LIN {X 0,Y 315.723,Z 316.79,A -85,B 0,C 180,E1 -15907.418,E2 -15907.418} C_VEL
LIN {X 0,Y 314.175,Z 327.926,A -85,B 0,C 180,E1 -15908.339,E2 -15908.339} C_VEL
LIN {X 0,Y 312.459,Z 339.529,A -85,B 0,C 180,E1 -15909.595,E2 -15909.595} C_VEL
LIN {X 0,Y 310.609,Z 350.036,A -85,B 0,C 180,E1 -15911.018,E2 -15911.018} C_VEL
LIN {X 0,Y 309.084,Z 358.664,A -85,B 0,C 180,E1 -15912.465,E2 -15912.465} C_VEL
LIN {X 0,Y 307.686,Z 366.655,A -85,B 0,C 180,E1 -15914.091,E2 -15914.091} C_VEL
LIN {X 0,Y 306.274,Z 374.524,A -85,B 0,C 180,E1 -15916.057,E2 -15916.057} C_VEL
LIN {X 0,Y 305.07,Z 380.86,A -85,B 0,C 180,E1 -15918.033,E2 -15918.033} C_VEL
LIN {X 0,Y 304.358,Z 385.924,A -85,B 0,C 180,E1 -15920.026,E2 -15920.026} C_VEL
LIN {X 0,Y 303.916,Z 389.858,A -85,B 0,C 180,E1 -15922.024,E2 -15922.024} C_VEL
LIN {X 0,Y 303.628,Z 393.261,A -85,B 0,C 180,E1 -15924.455,E2 -15924.455} C_VEL
LIN {X 0,Y 303.639,Z 394.706,A -85,B 0,C 180,E1 -15926.018,E2 -15926.018} C_VEL
LIN {X 0,Y 303.654,Z 395.466,A -85,B 0,C 180,E1 -15927.346,E2 -15927.346} C_VEL
LIN {X 0,Y 303.685,Z 395.832,A -85,B 0,C 180,E1 -15928.673,E2 -15928.673} C_VEL
LIN {X 0,Y 303.763,Z 395.804,A -85,B 0,C 180,E1 -15929.999,E2 -15929.999} C_VEL
LIN {X 0,Y 303.694,Z 395.325,A -85,B 0,C 180,E1 -15931.325,E2 -15931.325} C_VEL
LIN {X 0,Y 303.671,Z 394.427,A -85,B 0,C 180,E1 -15932.652,E2 -15932.652} C_VEL
LIN {X 0,Y 303.684,Z 393.121,A -85,B 0,C 180,E1 -15933.98,E2 -15933.98} C_VEL
LIN {X 0,Y 303.668,Z 390.884,A -85,B 0,C 180,E1 -15935.623,E2 -15935.623} C_VEL
LIN {X 0,Y 303.914,Z 386.438,A -85,B 0,C 180,E1 -15937.975,E2 -15937.975} C_VEL
LIN {X 0,Y 304.3,Z 381.396,A -85,B 0,C 180,E1 -15939.974,E2 -15939.974} C_VEL
LIN {X 0,Y 304.898,Z 375.03,A -85,B 0,C 180,E1 -15941.972,E2 -15941.972} C_VEL
LIN {X 0,Y 305.955,Z 367.045,A -85,B 0,C 180,E1 -15943.956,E2 -15943.956} C_VEL
LIN {X 0,Y 306.977,Z 358.879,A -85,B 0,C 180,E1 -15945.604,E2 -15945.604} C_VEL
LIN {X 0,Y 308.137,Z 348.901,A -85,B 0,C 180,E1 -15947.247,E2 -15947.247} C_VEL
LIN {X 0,Y 309.56,Z 337.739,A -85,B 0,C 180,E1 -15948.703,E2 -15948.703} C_VEL
LIN {X 0,Y 310.984,Z 325.048,A -85,B 0,C 180,E1 -15949.987,E2 -15949.987} C_VEL
LIN {X 0,Y 312.215,Z 312.461,A -85,B 0,C 180,E1 -15950.937,E2 -15950.937} C_VEL
LIN {X 0,Y 313.215,Z 299.169,A -85,B 0,C 180,E1 -15951.643,E2 -15951.643} C_VEL
LIN {X 0,Y 313.823,Z 286.404,A -85,B 0,C 180,E1 -15952.074,E2 -15952.074} C_VEL
LIN {X 0,Y 315.222,Z 226.259,A -85,B 0,C 180,E1 -15953.544,E2 -15953.544} C_VEL
LIN {X 0,Y 309.309,Z 183.433,A -85,B 0,C 180,E1 -15955.1,E2 -15955.1} C_VEL
LIN {X 0,Y 309.937,Z 177.619,A -85,B 0,C 180,E1 -15956.605,E2 -15956.605} C_VEL
LIN {X 0,Y 308.248,Z 168.036,A -85,B 0,C 180,E1 -15959.303,E2 -15959.303} C_VEL
LIN {X 0,Y 305.482,Z 155.435,A -85,B 0,C 180,E1 -15963.07,E2 -15963.07} C_VEL
LIN {X 0,Y 305.481,Z 155.431,A -85,B 0,C 180,E1 -15966.738,E2 -15966.738} C_VEL
LIN {X 0,Y 305.455,Z 155.435,A -85,B 0,C 180,E1 -15970.599,E2 -15970.599} C_VEL
LIN {X 0,Y 305.425,Z 155.442,A -85,B 0,C 180,E1 -15973.654,E2 -15973.654} C_VEL
LIN {X 0,Y 305.455,Z 155.436,A -85,B 0,C 180,E1 -15977.413,E2 -15977.413} C_VEL
LIN {X 0,Y 305.475,Z 155.436,A -85,B 0,C 180,E1 -15981.597,E2 -15981.597} C_VEL
LIN {X 0,Y 305.461,Z 155.433,A -85,B 0,C 180,E1 -15984.886,E2 -15984.886} C_VEL
LIN {X 0,Y 305.451,Z 155.434,A -85,B 0,C 180,E1 -15988.354,E2 -15988.354} C_VEL
LIN {X 0,Y 305.52,Z 155.427,A -85,B 0,C 180,E1 -15991.113,E2 -15991.113} C_VEL
LIN {X 0,Y 305.571,Z 155.419,A -85,B 0,C 180,E1 -15994.087,E2 -15994.087} C_VEL
LIN {X 0,Y 305.493,Z 155.429,A -85,B 0,C 180,E1 -15998.402,E2 -15998.402} C_VEL
LIN {X 0,Y 305.541,Z 155.428,A -85,B 0,C 180,E1 -16001.214,E2 -16001.214} C_VEL
LIN {X 0,Y 305.624,Z 155.416,A -85,B 0,C 180,E1 -16005.347,E2 -16005.347} C_VEL
LIN {X 0,Y 305.636,Z 155.412,A -85,B 0,C 180,E1 -16009.399,E2 -16009.399} C_VEL
LIN {X 0,Y 305.806,Z 155.387,A -85,B 0,C 180,E1 -16012.073,E2 -16012.073} C_VEL
LIN {X 0,Y 305.685,Z 155.407,A -85,B 0,C 180,E1 -16014.723,E2 -16014.723} C_VEL
LIN {X 0,Y 305.955,Z 155.375,A -85,B 0,C 180,E1 -16018.683,E2 -16018.683} C_VEL
LIN {X 0,Y 305.955,Z 155.37,A -85,B 0,C 180,E1 -16021.316,E2 -16021.316} C_VEL
LIN {X 0,Y 305.843,Z 155.389,A -85,B 0,C 180,E1 -16026.597,E2 -16026.597} C_VEL
LIN {X 0,Y 305.732,Z 155.399,A -85,B 0,C 180,E1 -16029.259,E2 -16029.259} C_VEL
LIN {X 0,Y 305.585,Z 155.414,A -85,B 0,C 180,E1 -16033.295,E2 -16033.295} C_VEL
LIN {X 0,Y 305.59,Z 155.416,A -85,B 0,C 180,E1 -16036.019,E2 -16036.019} C_VEL
LIN {X 0,Y 305.574,Z 155.418,A -85,B 0,C 180,E1 -16039.445,E2 -16039.445} C_VEL
LIN {X 0,Y 305.487,Z 155.428,A -85,B 0,C 180,E1 -16043.041,E2 -16043.041} C_VEL
LIN {X 0,Y 305.543,Z 155.423,A -85,B 0,C 180,E1 -16046.227,E2 -16046.227} C_VEL
LIN {X 0,Y 305.491,Z 155.428,A -85,B 0,C 180,E1 -16049.049,E2 -16049.049} C_VEL
LIN {X 0,Y 305.44,Z 155.438,A -85,B 0,C 180,E1 -16051.952,E2 -16051.952} C_VEL
LIN {X 0,Y 305.458,Z 155.43,A -85,B 0,C 180,E1 -16055.113,E2 -16055.113} C_VEL
LIN {X 0,Y 305.489,Z 155.429,A -85,B 0,C 180,E1 -16058.539,E2 -16058.539} C_VEL
LIN {X 0,Y 305.517,Z 155.425,A -85,B 0,C 180,E1 -16062.599,E2 -16062.599} C_VEL
LIN {X 0,Y 305.529,Z 155.424,A -85,B 0,C 180,E1 -16066.364,E2 -16066.364} C_VEL
LIN {X 0,Y 305.495,Z 155.433,A -85,B 0,C 180,E1 -16069.899,E2 -16069.899} C_VEL
LIN {X 0,Y 305.497,Z 155.432,A -85,B 0,C 180,E1 -16073.626,E2 -16073.626} C_VEL
LIN {X 0,Y 305.46,Z 155.433,A -85,B 0,C 180,E1 -16076.483,E2 -16076.483} C_VEL
LIN {X 0,Y 305.459,Z 155.438,A -85,B 0,C 180,E1 -16079.591,E2 -16079.591} C_VEL
LIN {X 0,Y 305.516,Z 155.426,A -85,B 0,C 180,E1 -16082.609,E2 -16082.609} C_VEL
LIN {X 0,Y 305.503,Z 155.432,A -85,B 0,C 180,E1 -16085.539,E2 -16085.539} C_VEL
LIN {X 0,Y 305.515,Z 155.428,A -85,B 0,C 180,E1 -16089.816,E2 -16089.816} C_VEL
LIN {X 0,Y 305.57,Z 155.42,A -85,B 0,C 180,E1 -16092.603,E2 -16092.603} C_VEL
LIN {X 0,Y 305.645,Z 155.415,A -85,B 0,C 180,E1 -16095.35,E2 -16095.35} C_VEL
LIN {X 0,Y 305.635,Z 155.415,A -85,B 0,C 180,E1 -16099.4,E2 -16099.4} C_VEL
LIN {X 0,Y 305.809,Z 155.39,A -85,B 0,C 180,E1 -16102.075,E2 -16102.075} C_VEL
LIN {X 0,Y 305.687,Z 155.407,A -85,B 0,C 180,E1 -16104.724,E2 -16104.724} C_VEL
LIN {X 0,Y 305.954,Z 155.374,A -85,B 0,C 180,E1 -16108.685,E2 -16108.685} C_VEL
LIN {X 0,Y 305.954,Z 155.374,A -85,B 0,C 180,E1 -16111.317,E2 -16111.317} C_VEL
LIN {X 0,Y 305.85,Z 155.388,A -85,B 0,C 180,E1 -16116.598,E2 -16116.598} C_VEL
LIN {X 0,Y 305.733,Z 155.401,A -85,B 0,C 180,E1 -16119.261,E2 -16119.261} C_VEL
LIN {X 0,Y 305.646,Z 155.427,A -85,B 0,C 180,E1 -16122.197,E2 -16122.197} C_VEL
LIN {X 0,Y 306.011,Z 157.364,A -85,B 0,C 180,E1 -16122.772,E2 -16122.772} C_VEL
LIN {X 0,Y 314.604,Z 181.076,A -85,B 0,C 180,E1 -16124.022,E2 -16124.022} C_VEL
LIN {X 0,Y 316.001,Z 185.936,A -85,B 0,C 180,E1 -16124.243,E2 -16124.243} C_VEL
LIN {X 0,Y 313.909,Z 265.333,A -85,B 0,C 180,E1 -16126.208,E2 -16126.208} C_VEL
LIN {X 0,Y 313.17,Z 279.059,A -85,B 0,C 180,E1 -16126.82,E2 -16126.82} C_VEL
LIN {X 0,Y 312.365,Z 291.964,A -85,B 0,C 180,E1 -16127.683,E2 -16127.683} C_VEL
LIN {X 0,Y 311.294,Z 304.537,A -85,B 0,C 180,E1 -16128.822,E2 -16128.822} C_VEL
LIN {X 0,Y 310.107,Z 315.16,A -85,B 0,C 180,E1 -16130.047,E2 -16130.047} C_VEL
LIN {X 0,Y 308.85,Z 325.402,A -85,B 0,C 180,E1 -16131.527,E2 -16131.527} C_VEL
LIN {X 0,Y 307.7,Z 334.503,A -85,B 0,C 180,E1 -16133.154,E2 -16133.154} C_VEL
LIN {X 0,Y 306.538,Z 343.308,A -85,B 0,C 180,E1 -16135.098,E2 -16135.098} C_VEL
LIN {X 0,Y 305.712,Z 349.648,A -85,B 0,C 180,E1 -16136.832,E2 -16136.832} C_VEL
LIN {X 0,Y 304.919,Z 355.858,A -85,B 0,C 180,E1 -16138.949,E2 -16138.949} C_VEL
LIN {X 0,Y 304.31,Z 361.08,A -85,B 0,C 180,E1 -16141.296,E2 -16141.296} C_VEL
LIN {X 0,Y 303.83,Z 364.938,A -85,B 0,C 180,E1 -16143.722,E2 -16143.722} C_VEL
LIN {X 0,Y 303.556,Z 367.113,A -85,B 0,C 180,E1 -16145.873,E2 -16145.873} C_VEL
LIN {X 0,Y 303.487,Z 368.209,A -85,B 0,C 180,E1 -16148.062,E2 -16148.062} C_VEL
LIN {X 0,Y 303.613,Z 368.161,A -85,B 0,C 180,E1 -16150.403,E2 -16150.403} C_VEL
LIN {X 0,Y 303.887,Z 367.26,A -85,B 0,C 180,E1 -16152.264,E2 -16152.264} C_VEL
LIN {X 0,Y 304.351,Z 365.346,A -85,B 0,C 180,E1 -16154.289,E2 -16154.289} C_VEL
LIN {X 0,Y 305.116,Z 361.546,A -85,B 0,C 180,E1 -16156.803,E2 -16156.803} C_VEL
LIN {X 0,Y 306.252,Z 356.287,A -85,B 0,C 180,E1 -16159.228,E2 -16159.228} C_VEL
LIN {X 0,Y 307.557,Z 349.621,A -85,B 0,C 180,E1 -16161.505,E2 -16161.505} C_VEL
LIN {X 0,Y 308.904,Z 342.905,A -85,B 0,C 180,E1 -16163.32,E2 -16163.32} C_VEL
LIN {X 0,Y 310.53,Z 334.566,A -85,B 0,C 180,E1 -16165.141,E2 -16165.141} C_VEL
LIN {X 0,Y 312.217,Z 325.27,A -85,B 0,C 180,E1 -16166.776,E2 -16166.776} C_VEL
LIN {X 0,Y 313.93,Z 314.467,A -85,B 0,C 180,E1 -16168.291,E2 -16168.291} C_VEL
LIN {X 0,Y 315.533,Z 303.485,A -85,B 0,C 180,E1 -16169.507,E2 -16169.507} C_VEL
LIN {X 0,Y 315.612,Z 298.386,A -85,B 0,C 180,E1 -16170.05,E2 -16170.05} C_VEL
LIN {X 0,Y 314.022,Z 290.018,A -85,B 0,C 180,E1 -16170.973,E2 -16170.973} C_VEL
LIN {X 0,Y 312.204,Z 281.348,A -85,B 0,C 180,E1 -16171.781,E2 -16171.781} C_VEL
LIN {X 0,Y 311.905,Z 275.779,A -85,B 0,C 180,E1 -16172.133,E2 -16172.133} C_VEL
LIN {X 0,Y 312.55,Z 264.777,A -85,B 0,C 180,E1 -16172.574,E2 -16172.574} C_VEL
LIN {X 0,Y 315.135,Z 192.637,A -85,B 0,C 180,E1 -16174.416,E2 -16174.416} C_VEL
LIN {X 0,Y 308.893,Z 177.993,A -85,B 0,C 180,E1 -16175.583,E2 -16175.583} C_VEL
LIN {X 0,Y 302.671,Z 165.931,A -85,B 0,C 180,E1 -16176.751,E2 -16176.751} C_VEL
LIN {X 0,Y 299.317,Z 159.58,A -85,B 0,C 180,E1 -16177.435,E2 -16177.435} C_VEL
LIN {X 0,Y 298.422,Z 156.314,A -85,B 0,C 180,E1 -16178.772,E2 -16178.772} C_VEL
LIN {X 0,Y 298.507,Z 156.301,A -85,B 0,C 180,E1 -16182.178,E2 -16182.178} C_VEL
LIN {X 0,Y 298.589,Z 156.293,A -85,B 0,C 180,E1 -16184.995,E2 -16184.995} C_VEL
LIN {X 0,Y 298.587,Z 156.292,A -85,B 0,C 180,E1 -16189.147,E2 -16189.147} C_VEL
LIN {X 0,Y 298.702,Z 156.279,A -85,B 0,C 180,E1 -16191.885,E2 -16191.885} C_VEL
LIN {X 0,Y 298.633,Z 156.287,A -85,B 0,C 180,E1 -16194.599,E2 -16194.599} C_VEL
LIN {X 0,Y 298.908,Z 156.245,A -85,B 0,C 180,E1 -16198.653,E2 -16198.653} C_VEL
LIN {X 0,Y 298.907,Z 156.252,A -85,B 0,C 180,E1 -16201.348,E2 -16201.348} C_VEL
LIN {X 0,Y 298.74,Z 156.26,A -85,B 0,C 180,E1 -16206.756,E2 -16206.756} C_VEL
LIN {X 0,Y 298.629,Z 156.286,A -85,B 0,C 180,E1 -16209.483,E2 -16209.483} C_VEL
LIN {X 0,Y 298.513,Z 156.299,A -85,B 0,C 180,E1 -16213.618,E2 -16213.618} C_VEL
LIN {X 0,Y 298.438,Z 156.306,A -85,B 0,C 180,E1 -16216.416,E2 -16216.416} C_VEL
LIN {X 0,Y 298.426,Z 156.301,A -85,B 0,C 180,E1 -16219.606,E2 -16219.606} C_VEL
LIN {X 0,Y 298.384,Z 156.307,A -85,B 0,C 180,E1 -16223.605,E2 -16223.605} C_VEL
LIN {X 0,Y 298.406,Z 156.312,A -85,B 0,C 180,E1 -16226.583,E2 -16226.583} C_VEL
LIN {X 0,Y 298.362,Z 156.32,A -85,B 0,C 180,E1 -16229.648,E2 -16229.648} C_VEL
LIN {X 0,Y 298.398,Z 156.313,A -85,B 0,C 180,E1 -16232.801,E2 -16232.801} C_VEL
LIN {X 0,Y 298.446,Z 156.311,A -85,B 0,C 180,E1 -16236.806,E2 -16236.806} C_VEL
LIN {X 0,Y 298.353,Z 156.317,A -85,B 0,C 180,E1 -16241.079,E2 -16241.079} C_VEL
LIN {X 0,Y 298.36,Z 156.325,A -85,B 0,C 180,E1 -16245.035,E2 -16245.035} C_VEL
LIN {X 0,Y 298.353,Z 156.322,A -85,B 0,C 180,E1 -16248.921,E2 -16248.921} C_VEL
LIN {X 0,Y 298.443,Z 156.429,A -85,B 0,C 180,E1 -16252.981,E2 -16252.981} C_VEL
LIN {X 0,Y 300.851,Z 165.427,A -85,B 0,C 180,E1 -16256.251,E2 -16256.251} C_VEL
LIN {X 0,Y 303.031,Z 174.547,A -85,B 0,C 180,E1 -16259.32,E2 -16259.32} C_VEL
LIN {X 0,Y 304.282,Z 180.764,A -85,B 0,C 180,E1 -16261.284,E2 -16261.284} C_VEL
LIN {X 0,Y 307.064,Z 187.661,A -85,B 0,C 180,E1 -16261.845,E2 -16261.845} C_VEL
LIN {X 0,Y 310.502,Z 204.648,A -85,B 0,C 180,E1 -16262.771,E2 -16262.771} C_VEL
LIN {X 0,Y 313.101,Z 221.424,A -85,B 0,C 180,E1 -16263.561,E2 -16263.561} C_VEL
LIN {X 0,Y 313.982,Z 230.204,A -85,B 0,C 180,E1 -16263.914,E2 -16263.914} C_VEL
LIN {X 0,Y 311.806,Z 291.118,A -85,B 0,C 180,E1 -16265.488,E2 -16265.488} C_VEL
LIN {X 0,Y 310.703,Z 305.109,A -85,B 0,C 180,E1 -16266.106,E2 -16266.106} C_VEL
LIN {X 0,Y 309.231,Z 317.646,A -85,B 0,C 180,E1 -16266.917,E2 -16266.917} C_VEL
LIN {X 0,Y 307.45,Z 330.063,A -85,B 0,C 180,E1 -16268.017,E2 -16268.017} C_VEL
LIN {X 0,Y 305.641,Z 341.228,A -85,B 0,C 180,E1 -16269.295,E2 -16269.295} C_VEL
LIN {X 0,Y 303.751,Z 351.344,A -85,B 0,C 180,E1 -16270.748,E2 -16270.748} C_VEL
LIN {X 0,Y 302.012,Z 360.519,A -85,B 0,C 180,E1 -16272.39,E2 -16272.39} C_VEL
LIN {X 0,Y 300.33,Z 369.507,A -85,B 0,C 180,E1 -16274.388,E2 -16274.388} C_VEL
LIN {X 0,Y 298.93,Z 376.767,A -85,B 0,C 180,E1 -16276.401,E2 -16276.401} C_VEL
LIN {X 0,Y 297.828,Z 382.586,A -85,B 0,C 180,E1 -16278.428,E2 -16278.428} C_VEL
LIN {X 0,Y 297.139,Z 387.208,A -85,B 0,C 180,E1 -16280.469,E2 -16280.469} C_VEL
LIN {X 0,Y 296.713,Z 390.748,A -85,B 0,C 180,E1 -16282.514,E2 -16282.514} C_VEL
LIN {X 0,Y 296.535,Z 393.286,A -85,B 0,C 180,E1 -16284.559,E2 -16284.559} C_VEL
LIN {X 0,Y 296.535,Z 394.428,A -85,B 0,C 180,E1 -16285.922,E2 -16285.922} C_VEL
LIN {X 0,Y 296.577,Z 395.17,A -85,B 0,C 180,E1 -16287.283,E2 -16287.283} C_VEL
LIN {X 0,Y 296.598,Z 395.515,A -85,B 0,C 180,E1 -16288.641,E2 -16288.641} C_VEL
LIN {X 0,Y 296.671,Z 395.458,A -85,B 0,C 180,E1 -16289.999,E2 -16289.999} C_VEL
LIN {X 0,Y 296.606,Z 394.943,A -85,B 0,C 180,E1 -16291.357,E2 -16291.357} C_VEL
LIN {X 0,Y 296.594,Z 394.023,A -85,B 0,C 180,E1 -16292.716,E2 -16292.716} C_VEL
LIN {X 0,Y 296.597,Z 392.694,A -85,B 0,C 180,E1 -16294.076,E2 -16294.076} C_VEL
LIN {X 0,Y 296.616,Z 389.835,A -85,B 0,C 180,E1 -16296.119,E2 -16296.119} C_VEL
LIN {X 0,Y 296.85,Z 385.909,A -85,B 0,C 180,E1 -16298.166,E2 -16298.166} C_VEL
LIN {X 0,Y 297.361,Z 379.828,A -85,B 0,C 180,E1 -16300.554,E2 -16300.554} C_VEL
LIN {X 0,Y 298.121,Z 373.12,A -85,B 0,C 180,E1 -16302.594,E2 -16302.594} C_VEL
LIN {X 0,Y 299.207,Z 364.774,A -85,B 0,C 180,E1 -16304.625,E2 -16304.625} C_VEL
LIN {X 0,Y 300.338,Z 355.816,A -85,B 0,C 180,E1 -16306.378,E2 -16306.378} C_VEL
LIN {X 0,Y 301.696,Z 345.618,A -85,B 0,C 180,E1 -16307.978,E2 -16307.978} C_VEL
LIN {X 0,Y 303.163,Z 333.703,A -85,B 0,C 180,E1 -16309.465,E2 -16309.465} C_VEL
LIN {X 0,Y 304.557,Z 321.737,A -85,B 0,C 180,E1 -16310.603,E2 -16310.603} C_VEL
LIN {X 0,Y 305.703,Z 309.357,A -85,B 0,C 180,E1 -16311.493,E2 -16311.493} C_VEL
LIN {X 0,Y 306.562,Z 296.715,A -85,B 0,C 180,E1 -16312.137,E2 -16312.137} C_VEL
LIN {X 0,Y 307.169,Z 282.226,A -85,B 0,C 180,E1 -16312.578,E2 -16312.578} C_VEL
LIN {X 0,Y 308.452,Z 226.602,A -85,B 0,C 180,E1 -16313.972,E2 -16313.972} C_VEL
LIN {X 0,Y 302.488,Z 183.168,A -85,B 0,C 180,E1 -16315.59,E2 -16315.59} C_VEL
LIN {X 0,Y 302.925,Z 178.248,A -85,B 0,C 180,E1 -16316.897,E2 -16316.897} C_VEL
LIN {X 0,Y 300.938,Z 167.767,A -85,B 0,C 180,E1 -16319.946,E2 -16319.946} C_VEL
LIN {X 0,Y 298.431,Z 156.313,A -85,B 0,C 180,E1 -16323.449,E2 -16323.449} C_VEL
LIN {X 0,Y 298.451,Z 156.307,A -85,B 0,C 180,E1 -16326.808,E2 -16326.808} C_VEL
LIN {X 0,Y 298.409,Z 156.314,A -85,B 0,C 180,E1 -16329.485,E2 -16329.485} C_VEL
LIN {X 0,Y 298.399,Z 156.314,A -85,B 0,C 180,E1 -16333.102,E2 -16333.102} C_VEL
LIN {X 0,Y 298.403,Z 156.312,A -85,B 0,C 180,E1 -16336.92,E2 -16336.92} C_VEL
LIN {X 0,Y 298.404,Z 156.313,A -85,B 0,C 180,E1 -16341.005,E2 -16341.005} C_VEL
LIN {X 0,Y 298.418,Z 156.313,A -85,B 0,C 180,E1 -16343.929,E2 -16343.929} C_VEL
LIN {X 0,Y 298.394,Z 156.315,A -85,B 0,C 180,E1 -16347.982,E2 -16347.982} C_VEL
LIN {X 0,Y 298.469,Z 156.305,A -85,B 0,C 180,E1 -16351.904,E2 -16351.904} C_VEL
LIN {X 0,Y 298.485,Z 156.303,A -85,B 0,C 180,E1 -16354.923,E2 -16354.923} C_VEL
LIN {X 0,Y 298.437,Z 156.313,A -85,B 0,C 180,E1 -16359.314,E2 -16359.314} C_VEL
LIN {X 0,Y 298.476,Z 156.302,A -85,B 0,C 180,E1 -16362.175,E2 -16362.175} C_VEL
LIN {X 0,Y 298.584,Z 156.291,A -85,B 0,C 180,E1 -16364.994,E2 -16364.994} C_VEL
LIN {X 0,Y 298.592,Z 156.292,A -85,B 0,C 180,E1 -16369.146,E2 -16369.146} C_VEL
LIN {X 0,Y 298.752,Z 156.265,A -85,B 0,C 180,E1 -16371.885,E2 -16371.885} C_VEL
LIN {X 0,Y 298.656,Z 156.281,A -85,B 0,C 180,E1 -16374.598,E2 -16374.598} C_VEL
LIN {X 0,Y 298.922,Z 156.25,A -85,B 0,C 180,E1 -16378.652,E2 -16378.652} C_VEL
LIN {X 0,Y 298.921,Z 156.245,A -85,B 0,C 180,E1 -16381.346,E2 -16381.346} C_VEL
LIN {X 0,Y 298.789,Z 156.269,A -85,B 0,C 180,E1 -16386.753,E2 -16386.753} C_VEL
LIN {X 0,Y 298.677,Z 156.277,A -85,B 0,C 180,E1 -16389.48,E2 -16389.48} C_VEL
LIN {X 0,Y 298.548,Z 156.289,A -85,B 0,C 180,E1 -16393.615,E2 -16393.615} C_VEL
LIN {X 0,Y 298.545,Z 156.296,A -85,B 0,C 180,E1 -16396.408,E2 -16396.408} C_VEL
LIN {X 0,Y 298.508,Z 156.299,A -85,B 0,C 180,E1 -16399.655,E2 -16399.655} C_VEL
LIN {X 0,Y 298.454,Z 156.304,A -85,B 0,C 180,E1 -16403.597,E2 -16403.597} C_VEL
LIN {X 0,Y 298.485,Z 156.302,A -85,B 0,C 180,E1 -16406.574,E2 -16406.574} C_VEL
LIN {X 0,Y 298.416,Z 156.31,A -85,B 0,C 180,E1 -16409.641,E2 -16409.641} C_VEL
LIN {X 0,Y 298.391,Z 156.312,A -85,B 0,C 180,E1 -16412.8,E2 -16412.8} C_VEL
LIN {X 0,Y 298.465,Z 156.301,A -85,B 0,C 180,E1 -16416.814,E2 -16416.814} C_VEL
LIN {X 0,Y 298.452,Z 156.305,A -85,B 0,C 180,E1 -16421.249,E2 -16421.249} C_VEL
LIN {X 0,Y 298.484,Z 156.299,A -85,B 0,C 180,E1 -16425.061,E2 -16425.061} C_VEL
LIN {X 0,Y 298.451,Z 156.305,A -85,B 0,C 180,E1 -16428.897,E2 -16428.897} C_VEL
LIN {X 0,Y 298.465,Z 156.304,A -85,B 0,C 180,E1 -16433.186,E2 -16433.186} C_VEL
LIN {X 0,Y 298.39,Z 156.314,A -85,B 0,C 180,E1 -16437.2,E2 -16437.2} C_VEL
LIN {X 0,Y 298.427,Z 156.309,A -85,B 0,C 180,E1 -16440.615,E2 -16440.615} C_VEL
LIN {X 0,Y 298.479,Z 156.307,A -85,B 0,C 180,E1 -16443.474,E2 -16443.474} C_VEL
LIN {X 0,Y 298.43,Z 156.309,A -85,B 0,C 180,E1 -16446.698,E2 -16446.698} C_VEL
LIN {X 0,Y 298.535,Z 156.296,A -85,B 0,C 180,E1 -16450.757,E2 -16450.757} C_VEL
LIN {X 0,Y 298.589,Z 156.292,A -85,B 0,C 180,E1 -16454.995,E2 -16454.995} C_VEL
LIN {X 0,Y 298.59,Z 156.294,A -85,B 0,C 180,E1 -16459.147,E2 -16459.147} C_VEL
LIN {X 0,Y 298.754,Z 156.269,A -85,B 0,C 180,E1 -16461.887,E2 -16461.887} C_VEL
LIN {X 0,Y 298.657,Z 156.282,A -85,B 0,C 180,E1 -16464.6,E2 -16464.6} C_VEL
LIN {X 0,Y 298.92,Z 156.25,A -85,B 0,C 180,E1 -16468.654,E2 -16468.654} C_VEL
LIN {X 0,Y 298.921,Z 156.25,A -85,B 0,C 180,E1 -16471.348,E2 -16471.348} C_VEL
LIN {X 0,Y 298.795,Z 156.268,A -85,B 0,C 180,E1 -16476.755,E2 -16476.755} C_VEL
LIN {X 0,Y 298.678,Z 156.28,A -85,B 0,C 180,E1 -16479.481,E2 -16479.481} C_VEL
LIN {X 0,Y 298.604,Z 156.465,A -85,B 0,C 180,E1 -16481.885,E2 -16481.885} C_VEL
LIN {X 0,Y 298.907,Z 157.765,A -85,B 0,C 180,E1 -16482.239,E2 -16482.239} C_VEL
LIN {X 0,Y 307.692,Z 181.814,A -85,B 0,C 180,E1 -16483.559,E2 -16483.559} C_VEL
LIN {X 0,Y 309.444,Z 187.449,A -85,B 0,C 180,E1 -16483.834,E2 -16483.834} C_VEL
LIN {X 0,Y 307.204,Z 264.994,A -85,B 0,C 180,E1 -16485.781,E2 -16485.781} C_VEL
LIN {X 0,Y 306.438,Z 278.893,A -85,B 0,C 180,E1 -16486.403,E2 -16486.403} C_VEL
LIN {X 0,Y 305.639,Z 291.188,A -85,B 0,C 180,E1 -16487.222,E2 -16487.222} C_VEL
LIN {X 0,Y 304.6,Z 303.395,A -85,B 0,C 180,E1 -16488.323,E2 -16488.323} C_VEL
LIN {X 0,Y 303.316,Z 314.744,A -85,B 0,C 180,E1 -16489.633,E2 -16489.633} C_VEL
LIN {X 0,Y 302.094,Z 324.416,A -85,B 0,C 180,E1 -16491.023,E2 -16491.023} C_VEL
LIN {X 0,Y 300.886,Z 333.684,A -85,B 0,C 180,E1 -16492.67,E2 -16492.67} C_VEL
LIN {X 0,Y 299.66,Z 342.905,A -85,B 0,C 180,E1 -16494.712,E2 -16494.712} C_VEL
LIN {X 0,Y 298.721,Z 349.824,A -85,B 0,C 180,E1 -16496.619,E2 -16496.619} C_VEL
LIN {X 0,Y 297.919,Z 355.737,A -85,B 0,C 180,E1 -16498.649,E2 -16498.649} C_VEL
LIN {X 0,Y 297.369,Z 360.088,A -85,B 0,C 180,E1 -16500.54,E2 -16500.54} C_VEL
LIN {X 0,Y 296.875,Z 364.287,A -85,B 0,C 180,E1 -16502.99,E2 -16502.99} C_VEL
LIN {X 0,Y 296.568,Z 366.335,A -85,B 0,C 180,E1 -16504.664,E2 -16504.664} C_VEL
LIN {X 0,Y 296.438,Z 367.717,A -85,B 0,C 180,E1 -16506.35,E2 -16506.35} C_VEL
LIN {X 0,Y 296.418,Z 368.595,A -85,B 0,C 180,E1 -16508.519,E2 -16508.519} C_VEL
LIN {X 0,Y 296.556,Z 368.451,A -85,B 0,C 180,E1 -16510.682,E2 -16510.682} C_VEL
LIN {X 0,Y 297.028,Z 366.898,A -85,B 0,C 180,E1 -16513.329,E2 -16513.329} C_VEL
LIN {X 0,Y 297.792,Z 363.71,A -85,B 0,C 180,E1 -16515.987,E2 -16515.987} C_VEL
LIN {X 0,Y 298.498,Z 360.434,A -85,B 0,C 180,E1 -16517.874,E2 -16517.874} C_VEL
LIN {X 0,Y 299.642,Z 355.066,A -85,B 0,C 180,E1 -16520.188,E2 -16520.188} C_VEL
LIN {X 0,Y 300.861,Z 349.567,A -85,B 0,C 180,E1 -16522.036,E2 -16522.036} C_VEL
LIN {X 0,Y 302.431,Z 342.185,A -85,B 0,C 180,E1 -16524.031,E2 -16524.031} C_VEL
LIN {X 0,Y 304.025,Z 334.282,A -85,B 0,C 180,E1 -16525.754,E2 -16525.754} C_VEL
LIN {X 0,Y 305.882,Z 324.255,A -85,B 0,C 180,E1 -16527.505,E2 -16527.505} C_VEL
LIN {X 0,Y 307.509,Z 314.576,A -85,B 0,C 180,E1 -16528.865,E2 -16528.865} C_VEL
LIN {X 0,Y 309.289,Z 302.642,A -85,B 0,C 180,E1 -16530.195,E2 -16530.195} C_VEL
LIN {X 0,Y 310.73,Z 289.888,A -85,B 0,C 180,E1 -16531.275,E2 -16531.275} C_VEL
LIN {X 0,Y 311.787,Z 277.709,A -85,B 0,C 180,E1 -16532.034,E2 -16532.034} C_VEL
LIN {X 0,Y 311.905,Z 275.779,A -85,B 0,C 180,E1 -16532.133,E2 -16532.133} C_VEL
LIN {X 0,Y 311.619,Z 270.11,A -85,B 0,C 180,E1 -16532.451,E2 -16532.451} C_VEL
LIN {X 0,Y 307.508,Z 252.608,A -85,B 0,C 180,E1 -16533.498,E2 -16533.498} C_VEL
LIN {X 0,Y 307.059,Z 247.821,A -85,B 0,C 180,E1 -16533.684,E2 -16533.684} C_VEL
LIN {X 0,Y 307.104,Z 245.879,A -85,B 0,C 180,E1 -16533.736,E2 -16533.736} C_VEL
LIN {X 0,Y 309.095,Z 194.644,A -85,B 0,C 180,E1 -16535.05,E2 -16535.05} C_VEL
LIN {X 0,Y 302.855,Z 180.204,A -85,B 0,C 180,E1 -16536.272,E2 -16536.272} C_VEL
LIN {X 0,Y 297.115,Z 169.053,A -85,B 0,C 180,E1 -16537.402,E2 -16537.402} C_VEL
LIN {X 0,Y 292.177,Z 160.065,A -85,B 0,C 180,E1 -16538.435,E2 -16538.435} C_VEL
LIN {X 0,Y 291.398,Z 157.19,A -85,B 0,C 180,E1 -16539.633,E2 -16539.633} C_VEL
LIN {X 0,Y 291.444,Z 157.183,A -85,B 0,C 180,E1 -16543.18,E2 -16543.18} C_VEL
LIN {X 0,Y 291.519,Z 157.177,A -85,B 0,C 180,E1 -16546.05,E2 -16546.05} C_VEL
LIN {X 0,Y 291.572,Z 157.167,A -85,B 0,C 180,E1 -16550.287,E2 -16550.287} C_VEL
LIN {X 0,Y 291.691,Z 157.151,A -85,B 0,C 180,E1 -16553.082,E2 -16553.082} C_VEL
LIN {X 0,Y 291.875,Z 157.121,A -85,B 0,C 180,E1 -16558.621,E2 -16558.621} C_VEL
LIN {X 0,Y 291.874,Z 157.128,A -85,B 0,C 180,E1 -16561.381,E2 -16561.381} C_VEL
LIN {X 0,Y 291.692,Z 157.138,A -85,B 0,C 180,E1 -16566.92,E2 -16566.92} C_VEL
LIN {X 0,Y 291.572,Z 157.161,A -85,B 0,C 180,E1 -16569.715,E2 -16569.715} C_VEL
LIN {X 0,Y 291.476,Z 157.172,A -85,B 0,C 180,E1 -16573.953,E2 -16573.953} C_VEL
LIN {X 0,Y 291.392,Z 157.185,A -85,B 0,C 180,E1 -16576.824,E2 -16576.824} C_VEL
LIN {X 0,Y 291.368,Z 157.181,A -85,B 0,C 180,E1 -16579.827,E2 -16579.827} C_VEL
LIN {X 0,Y 291.328,Z 157.187,A -85,B 0,C 180,E1 -16584.212,E2 -16584.212} C_VEL
LIN {X 0,Y 291.333,Z 157.187,A -85,B 0,C 180,E1 -16587.281,E2 -16587.281} C_VEL
LIN {X 0,Y 291.307,Z 157.197,A -85,B 0,C 180,E1 -16590.441,E2 -16590.441} C_VEL
LIN {X 0,Y 291.349,Z 157.193,A -85,B 0,C 180,E1 -16593.699,E2 -16593.699} C_VEL
LIN {X 0,Y 291.372,Z 157.189,A -85,B 0,C 180,E1 -16597.251,E2 -16597.251} C_VEL
LIN {X 0,Y 291.304,Z 157.197,A -85,B 0,C 180,E1 -16600.648,E2 -16600.648} C_VEL
LIN {X 0,Y 291.286,Z 157.201,A -85,B 0,C 180,E1 -16604.404,E2 -16604.404} C_VEL
LIN {X 0,Y 291.3,Z 157.202,A -85,B 0,C 180,E1 -16608.411,E2 -16608.411} C_VEL
LIN {X 0,Y 291.358,Z 157.293,A -85,B 0,C 180,E1 -16612.071,E2 -16612.071} C_VEL
LIN {X 0,Y 293.771,Z 165.928,A -85,B 0,C 180,E1 -16615.376,E2 -16615.376} C_VEL
LIN {X 0,Y 296.255,Z 176.398,A -85,B 0,C 180,E1 -16619.035,E2 -16619.035} C_VEL
LIN {X 0,Y 297.101,Z 180.321,A -85,B 0,C 180,E1 -16620.32,E2 -16620.32} C_VEL
LIN {X 0,Y 301.44,Z 190.585,A -85,B 0,C 180,E1 -16621.231,E2 -16621.231} C_VEL
LIN {X 0,Y 304.613,Z 206.594,A -85,B 0,C 180,E1 -16622.134,E2 -16622.134} C_VEL
LIN {X 0,Y 307.117,Z 223.332,A -85,B 0,C 180,E1 -16622.942,E2 -16622.942} C_VEL
LIN {X 0,Y 307.888,Z 231.171,A -85,B 0,C 180,E1 -16623.265,E2 -16623.265} C_VEL
LIN {X 0,Y 305.646,Z 290.506,A -85,B 0,C 180,E1 -16624.824,E2 -16624.824} C_VEL
LIN {X 0,Y 304.485,Z 304.521,A -85,B 0,C 180,E1 -16625.45,E2 -16625.45} C_VEL
LIN {X 0,Y 303.029,Z 316.591,A -85,B 0,C 180,E1 -16626.235,E2 -16626.235} C_VEL
LIN {X 0,Y 301.1,Z 329.132,A -85,B 0,C 180,E1 -16627.347,E2 -16627.347} C_VEL
LIN {X 0,Y 299.229,Z 340.365,A -85,B 0,C 180,E1 -16628.65,E2 -16628.65} C_VEL
LIN {X 0,Y 297.226,Z 350.59,A -85,B 0,C 180,E1 -16630.128,E2 -16630.128} C_VEL
LIN {X 0,Y 295.239,Z 360.661,A -85,B 0,C 180,E1 -16631.973,E2 -16631.973} C_VEL
LIN {X 0,Y 293.458,Z 369.574,A -85,B 0,C 180,E1 -16634.013,E2 -16634.013} C_VEL
LIN {X 0,Y 292.006,Z 376.739,A -85,B 0,C 180,E1 -16636.072,E2 -16636.072} C_VEL
LIN {X 0,Y 290.843,Z 382.495,A -85,B 0,C 180,E1 -16638.146,E2 -16638.146} C_VEL
LIN {X 0,Y 290.108,Z 387.056,A -85,B 0,C 180,E1 -16640.236,E2 -16640.236} C_VEL
LIN {X 0,Y 289.817,Z 389.483,A -85,B 0,C 180,E1 -16641.633,E2 -16641.633} C_VEL
LIN {X 0,Y 289.57,Z 391.478,A -85,B 0,C 180,E1 -16643.029,E2 -16643.029} C_VEL
LIN {X 0,Y 289.441,Z 393.176,A -85,B 0,C 180,E1 -16644.588,E2 -16644.588} C_VEL
LIN {X 0,Y 289.499,Z 394.874,A -85,B 0,C 180,E1 -16647.216,E2 -16647.216} C_VEL
LIN {X 0,Y 289.513,Z 395.199,A -85,B 0,C 180,E1 -16648.608,E2 -16648.608} C_VEL
LIN {X 0,Y 289.581,Z 395.103,A -85,B 0,C 180,E1 -16649.999,E2 -16649.999} C_VEL
LIN {X 0,Y 289.521,Z 394.562,A -85,B 0,C 180,E1 -16651.39,E2 -16651.39} C_VEL
LIN {X 0,Y 289.519,Z 393.62,A -85,B 0,C 180,E1 -16652.782,E2 -16652.782} C_VEL
LIN {X 0,Y 289.512,Z 392.266,A -85,B 0,C 180,E1 -16654.176,E2 -16654.176} C_VEL
LIN {X 0,Y 289.555,Z 389.359,A -85,B 0,C 180,E1 -16656.27,E2 -16656.27} C_VEL
LIN {X 0,Y 289.781,Z 385.379,A -85,B 0,C 180,E1 -16658.366,E2 -16658.366} C_VEL
LIN {X 0,Y 290.332,Z 379.211,A -85,B 0,C 180,E1 -16660.812,E2 -16660.812} C_VEL
LIN {X 0,Y 291.173,Z 372.439,A -85,B 0,C 180,E1 -16662.9,E2 -16662.9} C_VEL
LIN {X 0,Y 292.317,Z 364.015,A -85,B 0,C 180,E1 -16664.978,E2 -16664.978} C_VEL
LIN {X 0,Y 293.426,Z 355.317,A -85,B 0,C 180,E1 -16666.703,E2 -16666.703} C_VEL
LIN {X 0,Y 294.842,Z 344.593,A -85,B 0,C 180,E1 -16668.41,E2 -16668.41} C_VEL
LIN {X 0,Y 296.237,Z 333.98,A -85,B 0,C 180,E1 -16669.759,E2 -16669.759} C_VEL
LIN {X 0,Y 297.677,Z 322.234,A -85,B 0,C 180,E1 -16670.921,E2 -16670.921} C_VEL
LIN {X 0,Y 298.844,Z 310.095,A -85,B 0,C 180,E1 -16671.83,E2 -16671.83} C_VEL
LIN {X 0,Y 299.773,Z 297.017,A -85,B 0,C 180,E1 -16672.529,E2 -16672.529} C_VEL
LIN {X 0,Y 300.419,Z 283.01,A -85,B 0,C 180,E1 -16672.978,E2 -16672.978} C_VEL
LIN {X 0,Y 301.746,Z 227.294,A -85,B 0,C 180,E1 -16674.409,E2 -16674.409} C_VEL
LIN {X 0,Y 295.685,Z 182.895,A -85,B 0,C 180,E1 -16676.1,E2 -16676.1} C_VEL
LIN {X 0,Y 295.987,Z 180.255,A -85,B 0,C 180,E1 -16676.816,E2 -16676.816} C_VEL
LIN {X 0,Y 294.589,Z 171.875,A -85,B 0,C 180,E1 -16679.278,E2 -16679.278} C_VEL
LIN {X 0,Y 291.962,Z 159.672,A -85,B 0,C 180,E1 -16683.047,E2 -16683.047} C_VEL
LIN {X 0,Y 291.382,Z 157.19,A -85,B 0,C 180,E1 -16683.894,E2 -16683.894} C_VEL
LIN {X 0,Y 291.385,Z 157.188,A -85,B 0,C 180,E1 -16687.255,E2 -16687.255} C_VEL
LIN {X 0,Y 291.334,Z 157.195,A -85,B 0,C 180,E1 -16690.641,E2 -16690.641} C_VEL
LIN {X 0,Y 291.29,Z 157.2,A -85,B 0,C 180,E1 -16694.401,E2 -16694.401} C_VEL
LIN {X 0,Y 291.326,Z 157.194,A -85,B 0,C 180,E1 -16698.403,E2 -16698.403} C_VEL
LIN {X 0,Y 291.353,Z 157.192,A -85,B 0,C 180,E1 -16701.157,E2 -16701.157} C_VEL
LIN {X 0,Y 291.36,Z 157.19,A -85,B 0,C 180,E1 -16704.625,E2 -16704.625} C_VEL
LIN {X 0,Y 291.371,Z 157.19,A -85,B 0,C 180,E1 -16707.95,E2 -16707.95} C_VEL
LIN {X 0,Y 291.384,Z 157.187,A -85,B 0,C 180,E1 -16711.158,E2 -16711.158} C_VEL
LIN {X 0,Y 291.419,Z 157.182,A -85,B 0,C 180,E1 -16714.271,E2 -16714.271} C_VEL
LIN {X 0,Y 291.378,Z 157.19,A -85,B 0,C 180,E1 -16717.299,E2 -16717.299} C_VEL
LIN {X 0,Y 291.456,Z 157.177,A -85,B 0,C 180,E1 -16720.269,E2 -16720.269} C_VEL
LIN {X 0,Y 291.495,Z 157.171,A -85,B 0,C 180,E1 -16724.664,E2 -16724.664} C_VEL
LIN {X 0,Y 291.535,Z 157.171,A -85,B 0,C 180,E1 -16728.88,E2 -16728.88} C_VEL
LIN {X 0,Y 291.704,Z 157.143,A -85,B 0,C 180,E1 -16731.688,E2 -16731.688} C_VEL
LIN {X 0,Y 291.627,Z 157.155,A -85,B 0,C 180,E1 -16734.468,E2 -16734.468} C_VEL
LIN {X 0,Y 291.888,Z 157.126,A -85,B 0,C 180,E1 -16738.62,E2 -16738.62} C_VEL
LIN {X 0,Y 291.887,Z 157.12,A -85,B 0,C 180,E1 -16741.379,E2 -16741.379} C_VEL
LIN {X 0,Y 291.738,Z 157.145,A -85,B 0,C 180,E1 -16746.917,E2 -16746.917} C_VEL
LIN {X 0,Y 291.626,Z 157.156,A -85,B 0,C 180,E1 -16749.711,E2 -16749.711} C_VEL
LIN {X 0,Y 291.518,Z 157.165,A -85,B 0,C 180,E1 -16753.95,E2 -16753.95} C_VEL
LIN {X 0,Y 291.483,Z 157.175,A -85,B 0,C 180,E1 -16756.817,E2 -16756.817} C_VEL
LIN {X 0,Y 291.446,Z 157.179,A -85,B 0,C 180,E1 -16759.874,E2 -16759.874} C_VEL
LIN {X 0,Y 291.415,Z 157.183,A -85,B 0,C 180,E1 -16764.203,E2 -16764.203} C_VEL
LIN {X 0,Y 291.418,Z 157.178,A -85,B 0,C 180,E1 -16767.271,E2 -16767.271} C_VEL
LIN {X 0,Y 291.333,Z 157.195,A -85,B 0,C 180,E1 -16770.436,E2 -16770.436} C_VEL
LIN {X 0,Y 291.34,Z 157.191,A -85,B 0,C 180,E1 -16773.698,E2 -16773.698} C_VEL
LIN {X 0,Y 291.4,Z 157.18,A -85,B 0,C 180,E1 -16777.261,E2 -16777.261} C_VEL
LIN {X 0,Y 291.402,Z 157.184,A -85,B 0,C 180,E1 -16780.63,E2 -16780.63} C_VEL
LIN {X 0,Y 291.402,Z 157.183,A -85,B 0,C 180,E1 -16784.379,E2 -16784.379} C_VEL
LIN {X 0,Y 291.386,Z 157.186,A -85,B 0,C 180,E1 -16788.39,E2 -16788.39} C_VEL
LIN {X 0,Y 291.383,Z 157.187,A -85,B 0,C 180,E1 -16791.164,E2 -16791.164} C_VEL
LIN {X 0,Y 291.381,Z 157.184,A -85,B 0,C 180,E1 -16794.63,E2 -16794.63} C_VEL
LIN {X 0,Y 291.367,Z 157.191,A -85,B 0,C 180,E1 -16797.951,E2 -16797.951} C_VEL
LIN {X 0,Y 291.377,Z 157.189,A -85,B 0,C 180,E1 -16801.159,E2 -16801.159} C_VEL
LIN {X 0,Y 291.412,Z 157.183,A -85,B 0,C 180,E1 -16804.272,E2 -16804.272} C_VEL
LIN {X 0,Y 291.377,Z 157.191,A -85,B 0,C 180,E1 -16807.3,E2 -16807.3} C_VEL
LIN {X 0,Y 291.453,Z 157.178,A -85,B 0,C 180,E1 -16810.271,E2 -16810.271} C_VEL
LIN {X 0,Y 291.551,Z 157.167,A -85,B 0,C 180,E1 -16814.624,E2 -16814.624} C_VEL
LIN {X 0,Y 291.533,Z 157.171,A -85,B 0,C 180,E1 -16818.881,E2 -16818.881} C_VEL
LIN {X 0,Y 291.705,Z 157.148,A -85,B 0,C 180,E1 -16821.689,E2 -16821.689} C_VEL
LIN {X 0,Y 291.628,Z 157.158,A -85,B 0,C 180,E1 -16824.469,E2 -16824.469} C_VEL
LIN {X 0,Y 291.887,Z 157.126,A -85,B 0,C 180,E1 -16828.621,E2 -16828.621} C_VEL
LIN {X 0,Y 291.887,Z 157.126,A -85,B 0,C 180,E1 -16831.38,E2 -16831.38} C_VEL
LIN {X 0,Y 291.744,Z 157.147,A -85,B 0,C 180,E1 -16836.919,E2 -16836.919} C_VEL
LIN {X 0,Y 291.627,Z 157.158,A -85,B 0,C 180,E1 -16839.713,E2 -16839.713} C_VEL
LIN {X 0,Y 291.574,Z 157.355,A -85,B 0,C 180,E1 -16841.515,E2 -16841.515} C_VEL
LIN {X 0,Y 291.655,Z 157.842,A -85,B 0,C 180,E1 -16841.67,E2 -16841.67} C_VEL
LIN {X 0,Y 300.914,Z 182.888,A -85,B 0,C 180,E1 -16843.093,E2 -16843.093} C_VEL
LIN {X 0,Y 302.729,Z 188.356,A -85,B 0,C 180,E1 -16843.378,E2 -16843.378} C_VEL
LIN {X 0,Y 300.447,Z 266.048,A -85,B 0,C 180,E1 -16845.387,E2 -16845.387} C_VEL
LIN {X 0,Y 299.639,Z 280.06,A -85,B 0,C 180,E1 -16846.042,E2 -16846.042} C_VEL
LIN {X 0,Y 298.808,Z 292.578,A -85,B 0,C 180,E1 -16846.922,E2 -16846.922} C_VEL
LIN {X 0,Y 297.744,Z 304.25,A -85,B 0,C 180,E1 -16848.015,E2 -16848.015} C_VEL
LIN {X 0,Y 296.368,Z 315.805,A -85,B 0,C 180,E1 -16849.391,E2 -16849.391} C_VEL
LIN {X 0,Y 295.033,Z 326.043,A -85,B 0,C 180,E1 -16850.936,E2 -16850.936} C_VEL
LIN {X 0,Y 293.629,Z 336.364,A -85,B 0,C 180,E1 -16852.89,E2 -16852.89} C_VEL
LIN {X 0,Y 292.462,Z 344.768,A -85,B 0,C 180,E1 -16854.886,E2 -16854.886} C_VEL
LIN {X 0,Y 291.516,Z 351.485,A -85,B 0,C 180,E1 -16856.875,E2 -16856.875} C_VEL
LIN {X 0,Y 290.754,Z 357.001,A -85,B 0,C 180,E1 -16858.911,E2 -16858.911} C_VEL
LIN {X 0,Y 290.122,Z 361.933,A -85,B 0,C 180,E1 -16861.268,E2 -16861.268} C_VEL
LIN {X 0,Y 289.598,Z 365.852,A -85,B 0,C 180,E1 -16863.93,E2 -16863.93} C_VEL
LIN {X 0,Y 289.321,Z 368.239,A -85,B 0,C 180,E1 -16866.717,E2 -16866.717} C_VEL
LIN {X 0,Y 289.343,Z 369.008,A -85,B 0,C 180,E1 -16869.164,E2 -16869.164} C_VEL
LIN {X 0,Y 289.54,Z 368.674,A -85,B 0,C 180,E1 -16871.197,E2 -16871.197} C_VEL
LIN {X 0,Y 289.952,Z 367.394,A -85,B 0,C 180,E1 -16873.353,E2 -16873.353} C_VEL
LIN {X 0,Y 290.539,Z 365.191,A -85,B 0,C 180,E1 -16875.454,E2 -16875.454} C_VEL
LIN {X 0,Y 291.241,Z 362.1,A -85,B 0,C 180,E1 -16877.495,E2 -16877.495} C_VEL
LIN {X 0,Y 292.238,Z 358.016,A -85,B 0,C 180,E1 -16879.511,E2 -16879.511} C_VEL
LIN {X 0,Y 293.376,Z 352.945,A -85,B 0,C 180,E1 -16881.477,E2 -16881.477} C_VEL
LIN {X 0,Y 295.11,Z 345.374,A -85,B 0,C 180,E1 -16883.781,E2 -16883.781} C_VEL
LIN {X 0,Y 297.054,Z 336.36,A -85,B 0,C 180,E1 -16885.902,E2 -16885.902} C_VEL
LIN {X 0,Y 299.087,Z 326.344,A -85,B 0,C 180,E1 -16887.774,E2 -16887.774} C_VEL
LIN {X 0,Y 300.848,Z 316.546,A -85,B 0,C 180,E1 -16889.23,E2 -16889.23} C_VEL
LIN {X 0,Y 302.759,Z 304.54,A -85,B 0,C 180,E1 -16890.638,E2 -16890.638} C_VEL
LIN {X 0,Y 304.298,Z 292.328,A -85,B 0,C 180,E1 -16891.741,E2 -16891.741} C_VEL
LIN {X 0,Y 305.424,Z 279.467,A -85,B 0,C 180,E1 -16892.6,E2 -16892.6} C_VEL
LIN {X 0,Y 306.252,Z 267.398,A -85,B 0,C 180,E1 -16893.147,E2 -16893.147} C_VEL
LIN {X 0,Y 307.104,Z 245.879,A -85,B 0,C 180,E1 -16893.736,E2 -16893.736} C_VEL
LIN {X 0,Y 306.869,Z 240.089,A -85,B 0,C 180,E1 -16893.936,E2 -16893.936} C_VEL
LIN {X 0,Y 302.684,Z 221.519,A -85,B 0,C 180,E1 -16894.993,E2 -16894.993} C_VEL
LIN {X 0,Y 302.235,Z 215.737,A -85,B 0,C 180,E1 -16895.227,E2 -16895.227} C_VEL
LIN {X 0,Y 303.086,Z 196.669,A -85,B 0,C 180,E1 -16895.722,E2 -16895.722} C_VEL
LIN {X 0,Y 296.859,Z 182.282,A -85,B 0,C 180,E1 -16896.999,E2 -16896.999} C_VEL
LIN {X 0,Y 289.435,Z 168.215,A -85,B 0,C 180,E1 -16898.547,E2 -16898.547} C_VEL
LIN {X 0,Y 285.04,Z 160.498,A -85,B 0,C 180,E1 -16899.525,E2 -16899.525} C_VEL
LIN {X 0,Y 284.381,Z 158.06,A -85,B 0,C 180,E1 -16900.605,E2 -16900.605} C_VEL
LIN {X 0,Y 284.451,Z 158.052,A -85,B 0,C 180,E1 -16904.493,E2 -16904.493} C_VEL
LIN {X 0,Y 284.487,Z 158.053,A -85,B 0,C 180,E1 -16908.602,E2 -16908.602} C_VEL
LIN {X 0,Y 284.613,Z 158.037,A -85,B 0,C 180,E1 -16911.481,E2 -16911.481} C_VEL
LIN {X 0,Y 284.573,Z 158.042,A -85,B 0,C 180,E1 -16914.331,E2 -16914.331} C_VEL
LIN {X 0,Y 284.842,Z 157.997,A -85,B 0,C 180,E1 -16918.587,E2 -16918.587} C_VEL
LIN {X 0,Y 284.841,Z 158.005,A -85,B 0,C 180,E1 -16921.415,E2 -16921.415} C_VEL
LIN {X 0,Y 284.648,Z 158.015,A -85,B 0,C 180,E1 -16927.092,E2 -16927.092} C_VEL
LIN {X 0,Y 284.517,Z 158.037,A -85,B 0,C 180,E1 -16929.958,E2 -16929.958} C_VEL
LIN {X 0,Y 284.41,Z 158.049,A -85,B 0,C 180,E1 -16934.307,E2 -16934.307} C_VEL
LIN {X 0,Y 284.34,Z 158.065,A -85,B 0,C 180,E1 -16937.254,E2 -16937.254} C_VEL
LIN {X 0,Y 284.315,Z 158.062,A -85,B 0,C 180,E1 -16940.248,E2 -16940.248} C_VEL
LIN {X 0,Y 284.296,Z 158.062,A -85,B 0,C 180,E1 -16943.839,E2 -16943.839} C_VEL
LIN {X 0,Y 284.29,Z 158.065,A -85,B 0,C 180,E1 -16947.129,E2 -16947.129} C_VEL
LIN {X 0,Y 284.279,Z 158.073,A -85,B 0,C 180,E1 -16950.084,E2 -16950.084} C_VEL
LIN {X 0,Y 284.31,Z 158.069,A -85,B 0,C 180,E1 -16952.946,E2 -16952.946} C_VEL
LIN {X 0,Y 284.331,Z 158.067,A -85,B 0,C 180,E1 -16956.387,E2 -16956.387} C_VEL
LIN {X 0,Y 284.286,Z 158.074,A -85,B 0,C 180,E1 -16959.999,E2 -16959.999} C_VEL
LIN {X 0,Y 284.238,Z 158.078,A -85,B 0,C 180,E1 -16964.188,E2 -16964.188} C_VEL
LIN {X 0,Y 284.245,Z 158.082,A -85,B 0,C 180,E1 -16968.118,E2 -16968.118} C_VEL
LIN {X 0,Y 284.282,Z 158.191,A -85,B 0,C 180,E1 -16971.103,E2 -16971.103} C_VEL
LIN {X 0,Y 286.717,Z 166.471,A -85,B 0,C 180,E1 -16974.454,E2 -16974.454} C_VEL
LIN {X 0,Y 289.213,Z 176.931,A -85,B 0,C 180,E1 -16978.269,E2 -16978.269} C_VEL
LIN {X 0,Y 289.898,Z 179.93,A -85,B 0,C 180,E1 -16979.282,E2 -16979.282} C_VEL
LIN {X 0,Y 295.8,Z 193.157,A -85,B 0,C 180,E1 -16980.567,E2 -16980.567} C_VEL
LIN {X 0,Y 298.799,Z 208.826,A -85,B 0,C 180,E1 -16981.472,E2 -16981.472} C_VEL
LIN {X 0,Y 301.429,Z 226.807,A -85,B 0,C 180,E1 -16982.375,E2 -16982.375} C_VEL
LIN {X 0,Y 301.835,Z 232.017,A -85,B 0,C 180,E1 -16982.587,E2 -16982.587} C_VEL
LIN {X 0,Y 299.55,Z 289.893,A -85,B 0,C 180,E1 -16984.135,E2 -16984.135} C_VEL
LIN {X 0,Y 298.314,Z 303.988,A -85,B 0,C 180,E1 -16984.768,E2 -16984.768} C_VEL
LIN {X 0,Y 296.754,Z 316.617,A -85,B 0,C 180,E1 -16985.607,E2 -16985.607} C_VEL
LIN {X 0,Y 294.854,Z 328.291,A -85,B 0,C 180,E1 -16986.654,E2 -16986.654} C_VEL
LIN {X 0,Y 292.884,Z 339.615,A -85,B 0,C 180,E1 -16987.979,E2 -16987.979} C_VEL
LIN {X 0,Y 290.83,Z 349.908,A -85,B 0,C 180,E1 -16989.487,E2 -16989.487} C_VEL
LIN {X 0,Y 288.823,Z 359.201,A -85,B 0,C 180,E1 -16991.19,E2 -16991.19} C_VEL
LIN {X 0,Y 286.933,Z 368.273,A -85,B 0,C 180,E1 -16993.273,E2 -16993.273} C_VEL
LIN {X 0,Y 285.349,Z 375.638,A -85,B 0,C 180,E1 -16995.376,E2 -16995.376} C_VEL
LIN {X 0,Y 284.176,Z 380.644,A -85,B 0,C 180,E1 -16997.138,E2 -16997.138} C_VEL
LIN {X 0,Y 283.322,Z 385.537,A -85,B 0,C 180,E1 -16999.277,E2 -16999.277} C_VEL
LIN {X 0,Y 282.76,Z 389.314,A -85,B 0,C 180,E1 -17001.423,E2 -17001.423} C_VEL
LIN {X 0,Y 282.497,Z 391.285,A -85,B 0,C 180,E1 -17002.854,E2 -17002.854} C_VEL
LIN {X 0,Y 282.35,Z 393.105,A -85,B 0,C 180,E1 -17004.657,E2 -17004.657} C_VEL
LIN {X 0,Y 282.423,Z 394.582,A -85,B 0,C 180,E1 -17007.146,E2 -17007.146} C_VEL
LIN {X 0,Y 282.431,Z 394.882,A -85,B 0,C 180,E1 -17008.573,E2 -17008.573} C_VEL
LIN {X 0,Y 282.494,Z 394.741,A -85,B 0,C 180,E1 -17009.999,E2 -17009.999} C_VEL
LIN {X 0,Y 282.439,Z 394.178,A -85,B 0,C 180,E1 -17011.425,E2 -17011.425} C_VEL
LIN {X 0,Y 282.445,Z 393.215,A -85,B 0,C 180,E1 -17012.852,E2 -17012.852} C_VEL
LIN {X 0,Y 282.413,Z 391.832,A -85,B 0,C 180,E1 -17014.281,E2 -17014.281} C_VEL
LIN {X 0,Y 282.487,Z 388.882,A -85,B 0,C 180,E1 -17016.427,E2 -17016.427} C_VEL
LIN {X 0,Y 282.73,Z 384.848,A -85,B 0,C 180,E1 -17018.577,E2 -17018.577} C_VEL
LIN {X 0,Y 283.311,Z 378.593,A -85,B 0,C 180,E1 -17021.083,E2 -17021.083} C_VEL
LIN {X 0,Y 284.221,Z 371.755,A -85,B 0,C 180,E1 -17023.221,E2 -17023.221} C_VEL
LIN {X 0,Y 285.441,Z 363.234,A -85,B 0,C 180,E1 -17025.347,E2 -17025.347} C_VEL
LIN {X 0,Y 286.588,Z 354.412,A -85,B 0,C 180,E1 -17027.113,E2 -17027.113} C_VEL
LIN {X 0,Y 287.899,Z 344.752,A -85,B 0,C 180,E1 -17028.686,E2 -17028.686} C_VEL
LIN {X 0,Y 289.319,Z 334.234,A -85,B 0,C 180,E1 -17030.066,E2 -17030.066} C_VEL
LIN {X 0,Y 290.781,Z 322.701,A -85,B 0,C 180,E1 -17031.256,E2 -17031.256} C_VEL
LIN {X 0,Y 292.114,Z 309.527,A -85,B 0,C 180,E1 -17032.267,E2 -17032.267} C_VEL
LIN {X 0,Y 293.068,Z 296.343,A -85,B 0,C 180,E1 -17032.981,E2 -17032.981} C_VEL
LIN {X 0,Y 293.797,Z 280.489,A -85,B 0,C 180,E1 -17033.48,E2 -17033.48} C_VEL
LIN {X 0,Y 295.099,Z 228.124,A -85,B 0,C 180,E1 -17034.858,E2 -17034.858} C_VEL
LIN {X 0,Y 288.893,Z 182.595,A -85,B 0,C 180,E1 -17036.636,E2 -17036.636} C_VEL
LIN {X 0,Y 288.762,Z 179.452,A -85,B 0,C 180,E1 -17037.543,E2 -17037.543} C_VEL
LIN {X 0,Y 286.651,Z 168.541,A -85,B 0,C 180,E1 -17040.893,E2 -17040.893} C_VEL
LIN {X 0,Y 284.358,Z 158.065,A -85,B 0,C 180,E1 -17044.269,E2 -17044.269} C_VEL
LIN {X 0,Y 284.32,Z 158.07,A -85,B 0,C 180,E1 -17048.167,E2 -17048.167} C_VEL
LIN {X 0,Y 284.269,Z 158.077,A -85,B 0,C 180,E1 -17052.123,E2 -17052.123} C_VEL
LIN {X 0,Y 284.255,Z 158.076,A -85,B 0,C 180,E1 -17056.188,E2 -17056.188} C_VEL
LIN {X 0,Y 284.306,Z 158.07,A -85,B 0,C 180,E1 -17060.023,E2 -17060.023} C_VEL
LIN {X 0,Y 284.332,Z 158.07,A -85,B 0,C 180,E1 -17063.613,E2 -17063.613} C_VEL
LIN {X 0,Y 284.307,Z 158.071,A -85,B 0,C 180,E1 -17067.189,E2 -17067.189} C_VEL
LIN {X 0,Y 284.358,Z 158.059,A -85,B 0,C 180,E1 -17070.375,E2 -17070.375} C_VEL
LIN {X 0,Y 284.379,Z 158.062,A -85,B 0,C 180,E1 -17073.586,E2 -17073.586} C_VEL
LIN {X 0,Y 284.365,Z 158.059,A -85,B 0,C 180,E1 -17076.706,E2 -17076.706} C_VEL
LIN {X 0,Y 284.367,Z 158.064,A -85,B 0,C 180,E1 -17081.258,E2 -17081.258} C_VEL
LIN {X 0,Y 284.461,Z 158.049,A -85,B 0,C 180,E1 -17085.695,E2 -17085.695} C_VEL
LIN {X 0,Y 284.565,Z 158.035,A -85,B 0,C 180,E1 -17090.044,E2 -17090.044} C_VEL
LIN {X 0,Y 284.692,Z 158.02,A -85,B 0,C 180,E1 -17092.909,E2 -17092.909} C_VEL
LIN {X 0,Y 284.854,Z 158.002,A -85,B 0,C 180,E1 -17098.585,E2 -17098.585} C_VEL
LIN {X 0,Y 284.853,Z 157.996,A -85,B 0,C 180,E1 -17101.413,E2 -17101.413} C_VEL
LIN {X 0,Y 284.691,Z 158.022,A -85,B 0,C 180,E1 -17107.089,E2 -17107.089} C_VEL
LIN {X 0,Y 284.563,Z 158.036,A -85,B 0,C 180,E1 -17109.955,E2 -17109.955} C_VEL
LIN {X 0,Y 284.478,Z 158.043,A -85,B 0,C 180,E1 -17114.302,E2 -17114.302} C_VEL
LIN {X 0,Y 284.422,Z 158.053,A -85,B 0,C 180,E1 -17117.248,E2 -17117.248} C_VEL
LIN {X 0,Y 284.375,Z 158.062,A -85,B 0,C 180,E1 -17120.242,E2 -17120.242} C_VEL
LIN {X 0,Y 284.374,Z 158.058,A -85,B 0,C 180,E1 -17123.879,E2 -17123.879} C_VEL
LIN {X 0,Y 284.393,Z 158.053,A -85,B 0,C 180,E1 -17127.173,E2 -17127.173} C_VEL
LIN {X 0,Y 284.291,Z 158.069,A -85,B 0,C 180,E1 -17131.274,E2 -17131.274} C_VEL
LIN {X 0,Y 284.357,Z 158.057,A -85,B 0,C 180,E1 -17135.354,E2 -17135.354} C_VEL
LIN {X 0,Y 284.333,Z 158.066,A -85,B 0,C 180,E1 -17138.165,E2 -17138.165} C_VEL
LIN {X 0,Y 284.338,Z 158.067,A -85,B 0,C 180,E1 -17141.862,E2 -17141.862} C_VEL
LIN {X 0,Y 284.352,Z 158.062,A -85,B 0,C 180,E1 -17145.786,E2 -17145.786} C_VEL
LIN {X 0,Y 284.361,Z 158.064,A -85,B 0,C 180,E1 -17150.016,E2 -17150.016} C_VEL
LIN {X 0,Y 284.35,Z 158.065,A -85,B 0,C 180,E1 -17153.618,E2 -17153.618} C_VEL
LIN {X 0,Y 284.303,Z 158.069,A -85,B 0,C 180,E1 -17157.19,E2 -17157.19} C_VEL
LIN {X 0,Y 284.354,Z 158.062,A -85,B 0,C 180,E1 -17160.376,E2 -17160.376} C_VEL
LIN {X 0,Y 284.373,Z 158.064,A -85,B 0,C 180,E1 -17163.587,E2 -17163.587} C_VEL
LIN {X 0,Y 284.361,Z 158.061,A -85,B 0,C 180,E1 -17166.707,E2 -17166.707} C_VEL
LIN {X 0,Y 284.399,Z 158.061,A -85,B 0,C 180,E1 -17171.262,E2 -17171.262} C_VEL
LIN {X 0,Y 284.488,Z 158.046,A -85,B 0,C 180,E1 -17174.46,E2 -17174.46} C_VEL
LIN {X 0,Y 284.484,Z 158.048,A -85,B 0,C 180,E1 -17178.602,E2 -17178.602} C_VEL
LIN {X 0,Y 284.655,Z 158.028,A -85,B 0,C 180,E1 -17181.482,E2 -17181.482} C_VEL
LIN {X 0,Y 284.599,Z 158.033,A -85,B 0,C 180,E1 -17184.332,E2 -17184.332} C_VEL
LIN {X 0,Y 284.853,Z 158.002,A -85,B 0,C 180,E1 -17188.587,E2 -17188.587} C_VEL
LIN {X 0,Y 284.853,Z 158.002,A -85,B 0,C 180,E1 -17191.415,E2 -17191.415} C_VEL
LIN {X 0,Y 284.695,Z 158.024,A -85,B 0,C 180,E1 -17197.091,E2 -17197.091} C_VEL
LIN {X 0,Y 284.566,Z 158.038,A -85,B 0,C 180,E1 -17199.956,E2 -17199.956} C_VEL
LIN {X 0,Y 284.523,Z 158.108,A -85,B 0,C 180,E1 -17201.082,E2 -17201.082} C_VEL
LIN {X 0,Y 294.002,Z 183.533,A -85,B 0,C 180,E1 -17202.595,E2 -17202.595} C_VEL
LIN {X 0,Y 296.143,Z 190.293,A -85,B 0,C 180,E1 -17202.947,E2 -17202.947} C_VEL
LIN {X 0,Y 293.748,Z 266.177,A -85,B 0,C 180,E1 -17204.949,E2 -17204.949} C_VEL
LIN {X 0,Y 292.923,Z 279.762,A -85,B 0,C 180,E1 -17205.59,E2 -17205.59} C_VEL
LIN {X 0,Y 292.079,Z 292.186,A -85,B 0,C 180,E1 -17206.463,E2 -17206.463} C_VEL
LIN {X 0,Y 290.988,Z 303.936,A -85,B 0,C 180,E1 -17207.573,E2 -17207.573} C_VEL
LIN {X 0,Y 289.523,Z 315.97,A -85,B 0,C 180,E1 -17209.028,E2 -17209.028} C_VEL
LIN {X 0,Y 288.065,Z 326.867,A -85,B 0,C 180,E1 -17210.718,E2 -17210.718} C_VEL
LIN {X 0,Y 286.881,Z 335.271,A -85,B 0,C 180,E1 -17212.328,E2 -17212.328} C_VEL
LIN {X 0,Y 285.598,Z 344.188,A -85,B 0,C 180,E1 -17214.428,E2 -17214.428} C_VEL
LIN {X 0,Y 284.633,Z 350.872,A -85,B 0,C 180,E1 -17216.389,E2 -17216.389} C_VEL
LIN {X 0,Y 283.793,Z 356.581,A -85,B 0,C 180,E1 -17218.472,E2 -17218.472} C_VEL
LIN {X 0,Y 283.187,Z 361.133,A -85,B 0,C 180,E1 -17220.581,E2 -17220.581} C_VEL
LIN {X 0,Y 282.654,Z 365.221,A -85,B 0,C 180,E1 -17223.164,E2 -17223.164} C_VEL
LIN {X 0,Y 282.374,Z 367.204,A -85,B 0,C 180,E1 -17224.922,E2 -17224.922} C_VEL
LIN {X 0,Y 282.215,Z 368.777,A -85,B 0,C 180,E1 -17227.167,E2 -17227.167} C_VEL
LIN {X 0,Y 282.285,Z 369.345,A -85,B 0,C 180,E1 -17229.486,E2 -17229.486} C_VEL
LIN {X 0,Y 282.614,Z 368.655,A -85,B 0,C 180,E1 -17232.179,E2 -17232.179} C_VEL
LIN {X 0,Y 283.052,Z 367.364,A -85,B 0,C 180,E1 -17234.046,E2 -17234.046} C_VEL
LIN {X 0,Y 283.932,Z 363.927,A -85,B 0,C 180,E1 -17236.915,E2 -17236.915} C_VEL
LIN {X 0,Y 284.843,Z 360.439,A -85,B 0,C 180,E1 -17238.913,E2 -17238.913} C_VEL
LIN {X 0,Y 286.166,Z 354.909,A -85,B 0,C 180,E1 -17241.326,E2 -17241.326} C_VEL
LIN {X 0,Y 287.932,Z 347.854,A -85,B 0,C 180,E1 -17243.658,E2 -17243.658} C_VEL
LIN {X 0,Y 289.888,Z 339.303,A -85,B 0,C 180,E1 -17245.873,E2 -17245.873} C_VEL
LIN {X 0,Y 291.774,Z 330.706,A -85,B 0,C 180,E1 -17247.645,E2 -17247.645} C_VEL
LIN {X 0,Y 293.638,Z 321.456,A -85,B 0,C 180,E1 -17249.182,E2 -17249.182} C_VEL
LIN {X 0,Y 295.697,Z 309.954,A -85,B 0,C 180,E1 -17250.704,E2 -17250.704} C_VEL
LIN {X 0,Y 297.348,Z 298.688,A -85,B 0,C 180,E1 -17251.879,E2 -17251.879} C_VEL
LIN {X 0,Y 298.763,Z 285.753,A -85,B 0,C 180,E1 -17252.896,E2 -17252.896} C_VEL
LIN {X 0,Y 299.82,Z 272.47,A -85,B 0,C 180,E1 -17253.635,E2 -17253.635} C_VEL
LIN {X 0,Y 300.596,Z 257.803,A -85,B 0,C 180,E1 -17254.115,E2 -17254.115} C_VEL
LIN {X 0,Y 302.235,Z 215.737,A -85,B 0,C 180,E1 -17255.227,E2 -17255.227} C_VEL
LIN {X 0,Y 301.702,Z 209.98,A -85,B 0,C 180,E1 -17255.476,E2 -17255.476} C_VEL
LIN {X 0,Y 299.552,Z 202.791,A -85,B 0,C 180,E1 -17255.979,E2 -17255.979} C_VEL
LIN {X 0,Y 292.395,Z 187.666,A -85,B 0,C 180,E1 -17257.439,E2 -17257.439} C_VEL
LIN {X 0,Y 286.683,Z 176.335,A -85,B 0,C 180,E1 -17258.683,E2 -17258.683} C_VEL
LIN {X 0,Y 279.919,Z 164.582,A -85,B 0,C 180,E1 -17260.202,E2 -17260.202} C_VEL
LIN {X 0,Y 277.907,Z 160.912,A -85,B 0,C 180,E1 -17260.732,E2 -17260.732} C_VEL
LIN {X 0,Y 277.329,Z 158.941,A -85,B 0,C 180,E1 -17261.724,E2 -17261.724} C_VEL
LIN {X 0,Y 277.413,Z 158.933,A -85,B 0,C 180,E1 -17265.326,E2 -17265.326} C_VEL
LIN {X 0,Y 277.462,Z 158.923,A -85,B 0,C 180,E1 -17269.788,E2 -17269.788} C_VEL
LIN {X 0,Y 277.605,Z 158.904,A -85,B 0,C 180,E1 -17272.729,E2 -17272.729} C_VEL
LIN {X 0,Y 277.809,Z 158.873,A -85,B 0,C 180,E1 -17278.551,E2 -17278.551} C_VEL
LIN {X 0,Y 277.808,Z 158.881,A -85,B 0,C 180,E1 -17281.45,E2 -17281.45} C_VEL
LIN {X 0,Y 277.606,Z 158.892,A -85,B 0,C 180,E1 -17287.273,E2 -17287.273} C_VEL
LIN {X 0,Y 277.456,Z 158.914,A -85,B 0,C 180,E1 -17290.214,E2 -17290.214} C_VEL
LIN {X 0,Y 277.369,Z 158.923,A -85,B 0,C 180,E1 -17294.678,E2 -17294.678} C_VEL
LIN {X 0,Y 277.271,Z 158.936,A -85,B 0,C 180,E1 -17299.24,E2 -17299.24} C_VEL
LIN {X 0,Y 277.258,Z 158.938,A -85,B 0,C 180,E1 -17303.928,E2 -17303.928} C_VEL
LIN {X 0,Y 277.24,Z 158.941,A -85,B 0,C 180,E1 -17307.469,E2 -17307.469} C_VEL
LIN {X 0,Y 277.233,Z 158.949,A -85,B 0,C 180,E1 -17310.466,E2 -17310.466} C_VEL
LIN {X 0,Y 277.251,Z 158.948,A -85,B 0,C 180,E1 -17313.896,E2 -17313.896} C_VEL
LIN {X 0,Y 277.264,Z 158.945,A -85,B 0,C 180,E1 -17317.471,E2 -17317.471} C_VEL
LIN {X 0,Y 277.189,Z 158.953,A -85,B 0,C 180,E1 -17321.241,E2 -17321.241} C_VEL
LIN {X 0,Y 277.179,Z 158.964,A -85,B 0,C 180,E1 -17325.232,E2 -17325.232} C_VEL
LIN {X 0,Y 277.182,Z 158.959,A -85,B 0,C 180,E1 -17328.757,E2 -17328.757} C_VEL
LIN {X 0,Y 277.237,Z 159.021,A -85,B 0,C 180,E1 -17330.024,E2 -17330.024} C_VEL
LIN {X 0,Y 279.66,Z 167.246,A -85,B 0,C 180,E1 -17333.532,E2 -17333.532} C_VEL
LIN {X 0,Y 281.691,Z 175.456,A -85,B 0,C 180,E1 -17336.708,E2 -17336.708} C_VEL
LIN {X 0,Y 282.6,Z 179.377,A -85,B 0,C 180,E1 -17338.137,E2 -17338.137} C_VEL
LIN {X 0,Y 284.723,Z 183.786,A -85,B 0,C 180,E1 -17338.629,E2 -17338.629} C_VEL
LIN {X 0,Y 290.265,Z 195.95,A -85,B 0,C 180,E1 -17339.888,E2 -17339.888} C_VEL
LIN {X 0,Y 293.019,Z 210.677,A -85,B 0,C 180,E1 -17340.767,E2 -17340.767} C_VEL
LIN {X 0,Y 295.584,Z 228.903,A -85,B 0,C 180,E1 -17341.701,E2 -17341.701} C_VEL
LIN {X 0,Y 295.799,Z 234.019,A -85,B 0,C 180,E1 -17341.893,E2 -17341.893} C_VEL
LIN {X 0,Y 293.413,Z 290.522,A -85,B 0,C 180,E1 -17343.456,E2 -17343.456} C_VEL
LIN {X 0,Y 292.133,Z 304.248,A -85,B 0,C 180,E1 -17344.1,E2 -17344.1} C_VEL
LIN {X 0,Y 290.493,Z 316.634,A -85,B 0,C 180,E1 -17344.951,E2 -17344.951} C_VEL
LIN {X 0,Y 288.393,Z 329.018,A -85,B 0,C 180,E1 -17346.099,E2 -17346.099} C_VEL
LIN {X 0,Y 286.351,Z 340.154,A -85,B 0,C 180,E1 -17347.449,E2 -17347.449} C_VEL
LIN {X 0,Y 284.213,Z 350.255,A -85,B 0,C 180,E1 -17348.988,E2 -17348.988} C_VEL
LIN {X 0,Y 282.131,Z 359.424,A -85,B 0,C 180,E1 -17350.726,E2 -17350.726} C_VEL
LIN {X 0,Y 280.145,Z 368.407,A -85,B 0,C 180,E1 -17352.855,E2 -17352.855} C_VEL
LIN {X 0,Y 278.478,Z 375.671,A -85,B 0,C 180,E1 -17355.007,E2 -17355.007} C_VEL
LIN {X 0,Y 276.878,Z 382.328,A -85,B 0,C 180,E1 -17357.539,E2 -17357.539} C_VEL
LIN {X 0,Y 276.07,Z 386.77,A -85,B 0,C 180,E1 -17359.734,E2 -17359.734} C_VEL
LIN {X 0,Y 275.699,Z 389.146,A -85,B 0,C 180,E1 -17361.201,E2 -17361.201} C_VEL
LIN {X 0,Y 275.43,Z 391.08,A -85,B 0,C 180,E1 -17362.669,E2 -17362.669} C_VEL
LIN {X 0,Y 275.255,Z 393.044,A -85,B 0,C 180,E1 -17364.739,E2 -17364.739} C_VEL
LIN {X 0,Y 275.324,Z 394.291,A -85,B 0,C 180,E1 -17367.073,E2 -17367.073} C_VEL
LIN {X 0,Y 275.351,Z 394.555,A -85,B 0,C 180,E1 -17368.537,E2 -17368.537} C_VEL
LIN {X 0,Y 275.41,Z 394.374,A -85,B 0,C 180,E1 -17369.999,E2 -17369.999} C_VEL
LIN {X 0,Y 275.36,Z 393.787,A -85,B 0,C 180,E1 -17371.462,E2 -17371.462} C_VEL
LIN {X 0,Y 275.372,Z 392.798,A -85,B 0,C 180,E1 -17372.925,E2 -17372.925} C_VEL
LIN {X 0,Y 275.366,Z 389.975,A -85,B 0,C 180,E1 -17375.508,E2 -17375.508} C_VEL
LIN {X 0,Y 275.556,Z 385.736,A -85,B 0,C 180,E1 -17378.063,E2 -17378.063} C_VEL
LIN {X 0,Y 275.981,Z 380.85,A -85,B 0,C 180,E1 -17380.267,E2 -17380.267} C_VEL
LIN {X 0,Y 276.67,Z 374.653,A -85,B 0,C 180,E1 -17382.469,E2 -17382.469} C_VEL
LIN {X 0,Y 277.803,Z 366.936,A -85,B 0,C 180,E1 -17384.653,E2 -17384.653} C_VEL
LIN {X 0,Y 278.914,Z 359.38,A -85,B 0,C 180,E1 -17386.387,E2 -17386.387} C_VEL
LIN {X 0,Y 280.276,Z 349.298,A -85,B 0,C 180,E1 -17388.266,E2 -17388.266} C_VEL
LIN {X 0,Y 281.862,Z 338.564,A -85,B 0,C 180,E1 -17389.859,E2 -17389.859} C_VEL
LIN {X 0,Y 283.255,Z 328.212,A -85,B 0,C 180,E1 -17391.085,E2 -17391.085} C_VEL
LIN {X 0,Y 284.676,Z 315.893,A -85,B 0,C 180,E1 -17392.211,E2 -17392.211} C_VEL
LIN {X 0,Y 285.874,Z 303.084,A -85,B 0,C 180,E1 -17393.066,E2 -17393.066} C_VEL
LIN {X 0,Y 286.696,Z 289.679,A -85,B 0,C 180,E1 -17393.666,E2 -17393.666} C_VEL
LIN {X 0,Y 288.44,Z 228.972,A -85,B 0,C 180,E1 -17395.31,E2 -17395.31} C_VEL
LIN {X 0,Y 282.385,Z 184.167,A -85,B 0,C 180,E1 -17397.111,E2 -17397.111} C_VEL
LIN {X 0,Y 282.011,Z 182.191,A -85,B 0,C 180,E1 -17397.232,E2 -17397.232} C_VEL
LIN {X 0,Y 280.331,Z 172.988,A -85,B 0,C 180,E1 -17400.092,E2 -17400.092} C_VEL
LIN {X 0,Y 277.89,Z 161.597,A -85,B 0,C 180,E1 -17403.806,E2 -17403.806} C_VEL
LIN {X 0,Y 277.294,Z 158.945,A -85,B 0,C 180,E1 -17404.767,E2 -17404.767} C_VEL
LIN {X 0,Y 277.272,Z 158.948,A -85,B 0,C 180,E1 -17408.208,E2 -17408.208} C_VEL
LIN {X 0,Y 277.215,Z 158.954,A -85,B 0,C 180,E1 -17412.674,E2 -17412.674} C_VEL
LIN {X 0,Y 277.209,Z 158.953,A -85,B 0,C 180,E1 -17416.801,E2 -17416.801} C_VEL
LIN {X 0,Y 277.234,Z 158.949,A -85,B 0,C 180,E1 -17420.671,E2 -17420.671} C_VEL
LIN {X 0,Y 277.284,Z 158.944,A -85,B 0,C 180,E1 -17424.34,E2 -17424.34} C_VEL
LIN {X 0,Y 277.244,Z 158.951,A -85,B 0,C 180,E1 -17427.835,E2 -17427.835} C_VEL
LIN {X 0,Y 277.29,Z 158.943,A -85,B 0,C 180,E1 -17431.212,E2 -17431.212} C_VEL
LIN {X 0,Y 277.315,Z 158.939,A -85,B 0,C 180,E1 -17434.479,E2 -17434.479} C_VEL
LIN {X 0,Y 277.281,Z 158.945,A -85,B 0,C 180,E1 -17437.654,E2 -17437.654} C_VEL
LIN {X 0,Y 277.319,Z 158.94,A -85,B 0,C 180,E1 -17440.764,E2 -17440.764} C_VEL
LIN {X 0,Y 277.407,Z 158.93,A -85,B 0,C 180,E1 -17445.324,E2 -17445.324} C_VEL
LIN {X 0,Y 277.505,Z 158.914,A -85,B 0,C 180,E1 -17449.788,E2 -17449.788} C_VEL
LIN {X 0,Y 277.647,Z 158.895,A -85,B 0,C 180,E1 -17452.728,E2 -17452.728} C_VEL
LIN {X 0,Y 277.82,Z 158.878,A -85,B 0,C 180,E1 -17458.55,E2 -17458.55} C_VEL
LIN {X 0,Y 277.819,Z 158.871,A -85,B 0,C 180,E1 -17461.449,E2 -17461.449} C_VEL
LIN {X 0,Y 277.646,Z 158.899,A -85,B 0,C 180,E1 -17467.27,E2 -17467.27} C_VEL
LIN {X 0,Y 277.503,Z 158.916,A -85,B 0,C 180,E1 -17470.211,E2 -17470.211} C_VEL
LIN {X 0,Y 277.431,Z 158.923,A -85,B 0,C 180,E1 -17474.673,E2 -17474.673} C_VEL
LIN {X 0,Y 277.342,Z 158.935,A -85,B 0,C 180,E1 -17479.233,E2 -17479.233} C_VEL
LIN {X 0,Y 277.342,Z 158.935,A -85,B 0,C 180,E1 -17484.182,E2 -17484.182} C_VEL
LIN {X 0,Y 277.321,Z 158.934,A -85,B 0,C 180,E1 -17487.505,E2 -17487.505} C_VEL
LIN {X 0,Y 277.267,Z 158.946,A -85,B 0,C 180,E1 -17490.481,E2 -17490.481} C_VEL
LIN {X 0,Y 277.249,Z 158.947,A -85,B 0,C 180,E1 -17493.894,E2 -17493.894} C_VEL
LIN {X 0,Y 277.286,Z 158.937,A -85,B 0,C 180,E1 -17497.465,E2 -17497.465} C_VEL
LIN {X 0,Y 277.291,Z 158.941,A -85,B 0,C 180,E1 -17501.221,E2 -17501.221} C_VEL
LIN {X 0,Y 277.284,Z 158.939,A -85,B 0,C 180,E1 -17505.208,E2 -17505.208} C_VEL
LIN {X 0,Y 277.307,Z 158.941,A -85,B 0,C 180,E1 -17509.49,E2 -17509.49} C_VEL
LIN {X 0,Y 277.285,Z 158.942,A -85,B 0,C 180,E1 -17512.535,E2 -17512.535} C_VEL
LIN {X 0,Y 277.249,Z 158.948,A -85,B 0,C 180,E1 -17516.106,E2 -17516.106} C_VEL
LIN {X 0,Y 277.256,Z 158.951,A -85,B 0,C 180,E1 -17519.539,E2 -17519.539} C_VEL
LIN {X 0,Y 277.354,Z 158.935,A -85,B 0,C 180,E1 -17522.865,E2 -17522.865} C_VEL
LIN {X 0,Y 277.324,Z 158.938,A -85,B 0,C 180,E1 -17526.08,E2 -17526.08} C_VEL
LIN {X 0,Y 277.341,Z 158.937,A -85,B 0,C 180,E1 -17530.767,E2 -17530.767} C_VEL
LIN {X 0,Y 277.43,Z 158.93,A -85,B 0,C 180,E1 -17535.327,E2 -17535.327} C_VEL
LIN {X 0,Y 277.503,Z 158.918,A -85,B 0,C 180,E1 -17539.789,E2 -17539.789} C_VEL
LIN {X 0,Y 277.65,Z 158.9,A -85,B 0,C 180,E1 -17542.73,E2 -17542.73} C_VEL
LIN {X 0,Y 277.818,Z 158.878,A -85,B 0,C 180,E1 -17548.551,E2 -17548.551} C_VEL
LIN {X 0,Y 277.819,Z 158.878,A -85,B 0,C 180,E1 -17551.45,E2 -17551.45} C_VEL
LIN {X 0,Y 277.648,Z 158.9,A -85,B 0,C 180,E1 -17557.272,E2 -17557.272} C_VEL
LIN {X 0,Y 277.476,Z 158.923,A -85,B 0,C 180,E1 -17560.489,E2 -17560.489} C_VEL
LIN {X 0,Y 279.285,Z 163.688,A -85,B 0,C 180,E1 -17560.811,E2 -17560.811} C_VEL
LIN {X 0,Y 286.764,Z 183.422,A -85,B 0,C 180,E1 -17562.027,E2 -17562.027} C_VEL
LIN {X 0,Y 289.452,Z 191.387,A -85,B 0,C 180,E1 -17562.471,E2 -17562.471} C_VEL
LIN {X 0,Y 287.05,Z 266.151,A -85,B 0,C 180,E1 -17564.49,E2 -17564.49} C_VEL
LIN {X 0,Y 286.211,Z 279.863,A -85,B 0,C 180,E1 -17565.147,E2 -17565.147} C_VEL
LIN {X 0,Y 285.405,Z 291.291,A -85,B 0,C 180,E1 -17565.954,E2 -17565.954} C_VEL
LIN {X 0,Y 284.253,Z 303.515,A -85,B 0,C 180,E1 -17567.104,E2 -17567.104} C_VEL
LIN {X 0,Y 282.867,Z 314.772,A -85,B 0,C 180,E1 -17568.469,E2 -17568.469} C_VEL
LIN {X 0,Y 281.418,Z 325.159,A -85,B 0,C 180,E1 -17570.046,E2 -17570.046} C_VEL
LIN {X 0,Y 280.093,Z 334.513,A -85,B 0,C 180,E1 -17571.817,E2 -17571.817} C_VEL
LIN {X 0,Y 278.84,Z 342.911,A -85,B 0,C 180,E1 -17573.784,E2 -17573.784} C_VEL
LIN {X 0,Y 277.772,Z 350.152,A -85,B 0,C 180,E1 -17575.878,E2 -17575.878} C_VEL
LIN {X 0,Y 276.848,Z 356.256,A -85,B 0,C 180,E1 -17578.082,E2 -17578.082} C_VEL
LIN {X 0,Y 276.105,Z 361.624,A -85,B 0,C 180,E1 -17580.604,E2 -17580.604} C_VEL
LIN {X 0,Y 275.64,Z 364.99,A -85,B 0,C 180,E1 -17582.713,E2 -17582.713} C_VEL
LIN {X 0,Y 275.237,Z 367.734,A -85,B 0,C 180,E1 -17585.206,E2 -17585.206} C_VEL
LIN {X 0,Y 275.109,Z 369.312,A -85,B 0,C 180,E1 -17587.816,E2 -17587.816} C_VEL
LIN {X 0,Y 275.224,Z 369.651,A -85,B 0,C 180,E1 -17589.999,E2 -17589.999} C_VEL
LIN {X 0,Y 275.551,Z 369.041,A -85,B 0,C 180,E1 -17592.3,E2 -17592.3} C_VEL
LIN {X 0,Y 276.103,Z 367.477,A -85,B 0,C 180,E1 -17594.545,E2 -17594.545} C_VEL
LIN {X 0,Y 277.03,Z 364.11,A -85,B 0,C 180,E1 -17597.368,E2 -17597.368} C_VEL
LIN {X 0,Y 277.964,Z 360.732,A -85,B 0,C 180,E1 -17599.335,E2 -17599.335} C_VEL
LIN {X 0,Y 279.357,Z 355.344,A -85,B 0,C 180,E1 -17601.746,E2 -17601.746} C_VEL
LIN {X 0,Y 281.225,Z 348.235,A -85,B 0,C 180,E1 -17604.158,E2 -17604.158} C_VEL
LIN {X 0,Y 283.134,Z 340.359,A -85,B 0,C 180,E1 -17606.259,E2 -17606.259} C_VEL
LIN {X 0,Y 285.284,Z 331.208,A -85,B 0,C 180,E1 -17608.204,E2 -17608.204} C_VEL
LIN {X 0,Y 287.416,Z 320.832,A -85,B 0,C 180,E1 -17609.949,E2 -17609.949} C_VEL
LIN {X 0,Y 289.565,Z 309.506,A -85,B 0,C 180,E1 -17611.449,E2 -17611.449} C_VEL
LIN {X 0,Y 291.165,Z 298.983,A -85,B 0,C 180,E1 -17612.557,E2 -17612.557} C_VEL
LIN {X 0,Y 292.56,Z 287.128,A -85,B 0,C 180,E1 -17613.52,E2 -17613.52} C_VEL
LIN {X 0,Y 293.613,Z 274.942,A -85,B 0,C 180,E1 -17614.242,E2 -17614.242} C_VEL
LIN {X 0,Y 294.502,Z 261.695,A -85,B 0,C 180,E1 -17614.733,E2 -17614.733} C_VEL
LIN {X 0,Y 297.104,Z 198.591,A -85,B 0,C 180,E1 -17616.435,E2 -17616.435} C_VEL
LIN {X 0,Y 292.395,Z 187.666,A -85,B 0,C 180,E1 -17617.439,E2 -17617.439} C_VEL
LIN {X 0,Y 290.672,Z 184.624,A -85,B 0,C 180,E1 -17617.794,E2 -17617.794} C_VEL
LIN {X 0,Y 288.534,Z 182.023,A -85,B 0,C 180,E1 -17618.202,E2 -17618.202} C_VEL
LIN {X 0,Y 277.57,Z 172.229,A -85,B 0,C 180,E1 -17620.316,E2 -17620.316} C_VEL
LIN {X 0,Y 274.686,Z 168.097,A -85,B 0,C 180,E1 -17620.981,E2 -17620.981} C_VEL
LIN {X 0,Y 272.749,Z 164.966,A -85,B 0,C 180,E1 -17621.455,E2 -17621.455} C_VEL
LIN {X 0,Y 270.672,Z 161.377,A -85,B 0,C 180,E1 -17622.042,E2 -17622.042} C_VEL
LIN {X 0,Y 270.291,Z 159.816,A -85,B 0,C 180,E1 -17622.895,E2 -17622.895} C_VEL
LIN {X 0,Y 270.352,Z 159.811,A -85,B 0,C 180,E1 -17626.47,E2 -17626.47} C_VEL
LIN {X 0,Y 270.532,Z 159.793,A -85,B 0,C 180,E1 -17631.034,E2 -17631.034} C_VEL
LIN {X 0,Y 270.514,Z 159.793,A -85,B 0,C 180,E1 -17634.036,E2 -17634.036} C_VEL
LIN {X 0,Y 270.775,Z 159.75,A -85,B 0,C 180,E1 -17638.514,E2 -17638.514} C_VEL
LIN {X 0,Y 270.773,Z 159.757,A -85,B 0,C 180,E1 -17641.488,E2 -17641.488} C_VEL
LIN {X 0,Y 270.568,Z 159.77,A -85,B 0,C 180,E1 -17647.463,E2 -17647.463} C_VEL
LIN {X 0,Y 270.388,Z 159.792,A -85,B 0,C 180,E1 -17650.484,E2 -17650.484} C_VEL
LIN {X 0,Y 270.341,Z 159.797,A -85,B 0,C 180,E1 -17655.069,E2 -17655.069} C_VEL
LIN {X 0,Y 270.214,Z 159.815,A -85,B 0,C 180,E1 -17659.763,E2 -17659.763} C_VEL
LIN {X 0,Y 270.186,Z 159.821,A -85,B 0,C 180,E1 -17664.436,E2 -17664.436} C_VEL
LIN {X 0,Y 270.189,Z 159.819,A -85,B 0,C 180,E1 -17667.919,E2 -17667.919} C_VEL
LIN {X 0,Y 270.174,Z 159.822,A -85,B 0,C 180,E1 -17671.35,E2 -17671.35} C_VEL
LIN {X 0,Y 270.204,Z 159.82,A -85,B 0,C 180,E1 -17674.906,E2 -17674.906} C_VEL
LIN {X 0,Y 270.203,Z 159.821,A -85,B 0,C 180,E1 -17678.71,E2 -17678.71} C_VEL
LIN {X 0,Y 270.153,Z 159.835,A -85,B 0,C 180,E1 -17683.245,E2 -17683.245} C_VEL
LIN {X 0,Y 270.156,Z 159.839,A -85,B 0,C 180,E1 -17687.437,E2 -17687.437} C_VEL
LIN {X 0,Y 270.153,Z 159.88,A -85,B 0,C 180,E1 -17688.849,E2 -17688.849} C_VEL
LIN {X 0,Y 272.909,Z 169.026,A -85,B 0,C 180,E1 -17692.971,E2 -17692.971} C_VEL
LIN {X 0,Y 274.965,Z 177.406,A -85,B 0,C 180,E1 -17696.328,E2 -17696.328} C_VEL
LIN {X 0,Y 275.409,Z 179.131,A -85,B 0,C 180,E1 -17696.92,E2 -17696.92} C_VEL
LIN {X 0,Y 281.996,Z 192.555,A -85,B 0,C 180,E1 -17698.516,E2 -17698.516} C_VEL
LIN {X 0,Y 285.106,Z 200.127,A -85,B 0,C 180,E1 -17699.266,E2 -17699.266} C_VEL
LIN {X 0,Y 288.256,Z 218.713,A -85,B 0,C 180,E1 -17700.378,E2 -17700.378} C_VEL
LIN {X 0,Y 289.964,Z 233.414,A -85,B 0,C 180,E1 -17701.105,E2 -17701.105} C_VEL
LIN {X 0,Y 287.505,Z 289.313,A -85,B 0,C 180,E1 -17702.67,E2 -17702.67} C_VEL
LIN {X 0,Y 286.151,Z 303.303,A -85,B 0,C 180,E1 -17703.32,E2 -17703.32} C_VEL
LIN {X 0,Y 284.476,Z 315.877,A -85,B 0,C 180,E1 -17704.187,E2 -17704.187} C_VEL
LIN {X 0,Y 282.29,Z 328.306,A -85,B 0,C 180,E1 -17705.353,E2 -17705.353} C_VEL
LIN {X 0,Y 280.074,Z 339.478,A -85,B 0,C 180,E1 -17706.719,E2 -17706.719} C_VEL
LIN {X 0,Y 277.829,Z 349.626,A -85,B 0,C 180,E1 -17708.286,E2 -17708.286} C_VEL
LIN {X 0,Y 275.433,Z 359.65,A -85,B 0,C 180,E1 -17710.239,E2 -17710.239} C_VEL
LIN {X 0,Y 273.373,Z 368.543,A -85,B 0,C 180,E1 -17712.417,E2 -17712.417} C_VEL
LIN {X 0,Y 271.623,Z 375.696,A -85,B 0,C 180,E1 -17714.62,E2 -17714.62} C_VEL
LIN {X 0,Y 269.927,Z 382.279,A -85,B 0,C 180,E1 -17717.213,E2 -17717.213} C_VEL
LIN {X 0,Y 269.041,Z 386.655,A -85,B 0,C 180,E1 -17719.463,E2 -17719.463} C_VEL
LIN {X 0,Y 268.661,Z 388.995,A -85,B 0,C 180,E1 -17720.969,E2 -17720.969} C_VEL
LIN {X 0,Y 268.353,Z 390.871,A -85,B 0,C 180,E1 -17722.475,E2 -17722.475} C_VEL
LIN {X 0,Y 268.171,Z 392.943,A -85,B 0,C 180,E1 -17724.799,E2 -17724.799} C_VEL
LIN {X 0,Y 268.229,Z 394,A -85,B 0,C 180,E1 -17726.995,E2 -17726.995} C_VEL
LIN {X 0,Y 268.273,Z 394.216,A -85,B 0,C 180,E1 -17728.498,E2 -17728.498} C_VEL
LIN {X 0,Y 268.328,Z 394.009,A -85,B 0,C 180,E1 -17729.999,E2 -17729.999} C_VEL
LIN {X 0,Y 268.283,Z 393.396,A -85,B 0,C 180,E1 -17731.5,E2 -17731.5} C_VEL
LIN {X 0,Y 268.299,Z 392.381,A -85,B 0,C 180,E1 -17733.002,E2 -17733.002} C_VEL
LIN {X 0,Y 268.269,Z 389.791,A -85,B 0,C 180,E1 -17735.425,E2 -17735.425} C_VEL
LIN {X 0,Y 268.408,Z 386.572,A -85,B 0,C 180,E1 -17737.522,E2 -17737.522} C_VEL
LIN {X 0,Y 268.776,Z 382.028,A -85,B 0,C 180,E1 -17739.785,E2 -17739.785} C_VEL
LIN {X 0,Y 269.556,Z 375.089,A -85,B 0,C 180,E1 -17742.42,E2 -17742.42} C_VEL
LIN {X 0,Y 270.696,Z 367.535,A -85,B 0,C 180,E1 -17744.662,E2 -17744.662} C_VEL
LIN {X 0,Y 271.861,Z 359.812,A -85,B 0,C 180,E1 -17746.52,E2 -17746.52} C_VEL
LIN {X 0,Y 273.234,Z 350.416,A -85,B 0,C 180,E1 -17748.365,E2 -17748.365} C_VEL
LIN {X 0,Y 274.806,Z 339.967,A -85,B 0,C 180,E1 -17750.001,E2 -17750.001} C_VEL
LIN {X 0,Y 276.386,Z 328.397,A -85,B 0,C 180,E1 -17751.439,E2 -17751.439} C_VEL
LIN {X 0,Y 277.84,Z 316.284,A -85,B 0,C 180,E1 -17752.591,E2 -17752.591} C_VEL
LIN {X 0,Y 279.121,Z 302.968,A -85,B 0,C 180,E1 -17753.51,E2 -17753.51} C_VEL
LIN {X 0,Y 279.977,Z 289.755,A -85,B 0,C 180,E1 -17754.122,E2 -17754.122} C_VEL
LIN {X 0,Y 281.776,Z 229.354,A -85,B 0,C 180,E1 -17755.801,E2 -17755.801} C_VEL
LIN {X 0,Y 275.833,Z 185.556,A -85,B 0,C 180,E1 -17757.619,E2 -17757.619} C_VEL
LIN {X 0,Y 274.829,Z 181.892,A -85,B 0,C 180,E1 -17757.841,E2 -17757.841} C_VEL
LIN {X 0,Y 272.944,Z 172.096,A -85,B 0,C 180,E1 -17760.995,E2 -17760.995} C_VEL
LIN {X 0,Y 270.272,Z 159.82,A -85,B 0,C 180,E1 -17765.178,E2 -17765.178} C_VEL
LIN {X 0,Y 270.198,Z 159.827,A -85,B 0,C 180,E1 -17768.709,E2 -17768.709} C_VEL
LIN {X 0,Y 270.172,Z 159.832,A -85,B 0,C 180,E1 -17772.557,E2 -17772.557} C_VEL
LIN {X 0,Y 270.165,Z 159.83,A -85,B 0,C 180,E1 -17776.75,E2 -17776.75} C_VEL
LIN {X 0,Y 270.174,Z 159.831,A -85,B 0,C 180,E1 -17779.433,E2 -17779.433} C_VEL
LIN {X 0,Y 270.225,Z 159.826,A -85,B 0,C 180,E1 -17783.729,E2 -17783.729} C_VEL
LIN {X 0,Y 270.202,Z 159.826,A -85,B 0,C 180,E1 -17786.892,E2 -17786.892} C_VEL
LIN {X 0,Y 270.229,Z 159.819,A -85,B 0,C 180,E1 -17790.386,E2 -17790.386} C_VEL
LIN {X 0,Y 270.265,Z 159.819,A -85,B 0,C 180,E1 -17793.763,E2 -17793.763} C_VEL
LIN {X 0,Y 270.23,Z 159.821,A -85,B 0,C 180,E1 -17797.038,E2 -17797.038} C_VEL
LIN {X 0,Y 270.269,Z 159.817,A -85,B 0,C 180,E1 -17800.241,E2 -17800.241} C_VEL
LIN {X 0,Y 270.366,Z 159.804,A -85,B 0,C 180,E1 -17804.932,E2 -17804.932} C_VEL
LIN {X 0,Y 270.44,Z 159.795,A -85,B 0,C 180,E1 -17809.518,E2 -17809.518} C_VEL
LIN {X 0,Y 270.606,Z 159.771,A -85,B 0,C 180,E1 -17812.538,E2 -17812.538} C_VEL
LIN {X 0,Y 270.785,Z 159.754,A -85,B 0,C 180,E1 -17818.512,E2 -17818.512} C_VEL
LIN {X 0,Y 270.785,Z 159.747,A -85,B 0,C 180,E1 -17821.486,E2 -17821.486} C_VEL
LIN {X 0,Y 270.605,Z 159.775,A -85,B 0,C 180,E1 -17827.46,E2 -17827.46} C_VEL
LIN {X 0,Y 270.438,Z 159.798,A -85,B 0,C 180,E1 -17830.48,E2 -17830.48} C_VEL
LIN {X 0,Y 270.399,Z 159.797,A -85,B 0,C 180,E1 -17835.064,E2 -17835.064} C_VEL
LIN {X 0,Y 270.298,Z 159.813,A -85,B 0,C 180,E1 -17839.755,E2 -17839.755} C_VEL
LIN {X 0,Y 270.278,Z 159.809,A -85,B 0,C 180,E1 -17844.584,E2 -17844.584} C_VEL
LIN {X 0,Y 270.267,Z 159.814,A -85,B 0,C 180,E1 -17847.908,E2 -17847.908} C_VEL
LIN {X 0,Y 270.18,Z 159.826,A -85,B 0,C 180,E1 -17851.348,E2 -17851.348} C_VEL
LIN {X 0,Y 270.211,Z 159.818,A -85,B 0,C 180,E1 -17854.903,E2 -17854.903} C_VEL
LIN {X 0,Y 270.248,Z 159.817,A -85,B 0,C 180,E1 -17858.725,E2 -17858.725} C_VEL
LIN {X 0,Y 270.252,Z 159.818,A -85,B 0,C 180,E1 -17862.541,E2 -17862.541} C_VEL
LIN {X 0,Y 270.228,Z 159.817,A -85,B 0,C 180,E1 -17866.735,E2 -17866.735} C_VEL
LIN {X 0,Y 270.26,Z 159.818,A -85,B 0,C 180,E1 -17869.451,E2 -17869.451} C_VEL
LIN {X 0,Y 270.253,Z 159.819,A -85,B 0,C 180,E1 -17873.721,E2 -17873.721} C_VEL
LIN {X 0,Y 270.199,Z 159.825,A -85,B 0,C 180,E1 -17876.893,E2 -17876.893} C_VEL
LIN {X 0,Y 270.224,Z 159.822,A -85,B 0,C 180,E1 -17880.387,E2 -17880.387} C_VEL
LIN {X 0,Y 270.259,Z 159.821,A -85,B 0,C 180,E1 -17883.764,E2 -17883.764} C_VEL
LIN {X 0,Y 270.228,Z 159.823,A -85,B 0,C 180,E1 -17887.039,E2 -17887.039} C_VEL
LIN {X 0,Y 270.297,Z 159.814,A -85,B 0,C 180,E1 -17890.245,E2 -17890.245} C_VEL
LIN {X 0,Y 270.399,Z 159.804,A -85,B 0,C 180,E1 -17894.936,E2 -17894.936} C_VEL
LIN {X 0,Y 270.438,Z 159.8,A -85,B 0,C 180,E1 -17899.52,E2 -17899.52} C_VEL
LIN {X 0,Y 270.608,Z 159.777,A -85,B 0,C 180,E1 -17902.54,E2 -17902.54} C_VEL
LIN {X 0,Y 270.784,Z 159.755,A -85,B 0,C 180,E1 -17908.514,E2 -17908.514} C_VEL
LIN {X 0,Y 270.784,Z 159.754,A -85,B 0,C 180,E1 -17911.488,E2 -17911.488} C_VEL
LIN {X 0,Y 270.606,Z 159.777,A -85,B 0,C 180,E1 -17917.462,E2 -17917.462} C_VEL
LIN {X 0,Y 270.5,Z 159.79,A -85,B 0,C 180,E1 -17919.894,E2 -17919.894} C_VEL
LIN {X 0,Y 272.041,Z 164.091,A -85,B 0,C 180,E1 -17920.187,E2 -17920.187} C_VEL
LIN {X 0,Y 278.321,Z 179.825,A -85,B 0,C 180,E1 -17921.219,E2 -17921.219} C_VEL
LIN {X 0,Y 282.766,Z 192.66,A -85,B 0,C 180,E1 -17921.977,E2 -17921.977} C_VEL
LIN {X 0,Y 280.342,Z 266.726,A -85,B 0,C 180,E1 -17924.033,E2 -17924.033} C_VEL
LIN {X 0,Y 279.518,Z 279.908,A -85,B 0,C 180,E1 -17924.679,E2 -17924.679} C_VEL
LIN {X 0,Y 278.639,Z 291.92,A -85,B 0,C 180,E1 -17925.546,E2 -17925.546} C_VEL
LIN {X 0,Y 277.424,Z 304.282,A -85,B 0,C 180,E1 -17926.749,E2 -17926.749} C_VEL
LIN {X 0,Y 275.936,Z 315.683,A -85,B 0,C 180,E1 -17928.175,E2 -17928.175} C_VEL
LIN {X 0,Y 274.434,Z 326.22,A -85,B 0,C 180,E1 -17929.836,E2 -17929.836} C_VEL
LIN {X 0,Y 273.028,Z 335.684,A -85,B 0,C 180,E1 -17931.711,E2 -17931.711} C_VEL
LIN {X 0,Y 271.808,Z 343.574,A -85,B 0,C 180,E1 -17933.628,E2 -17933.628} C_VEL
LIN {X 0,Y 270.672,Z 350.972,A -85,B 0,C 180,E1 -17935.845,E2 -17935.845} C_VEL
LIN {X 0,Y 269.79,Z 356.632,A -85,B 0,C 180,E1 -17937.964,E2 -17937.964} C_VEL
LIN {X 0,Y 269.058,Z 361.834,A -85,B 0,C 180,E1 -17940.462,E2 -17940.462} C_VEL
LIN {X 0,Y 268.467,Z 365.823,A -85,B 0,C 180,E1 -17943.103,E2 -17943.103} C_VEL
LIN {X 0,Y 268.104,Z 368.376,A -85,B 0,C 180,E1 -17945.648,E2 -17945.648} C_VEL
LIN {X 0,Y 268.029,Z 369.714,A -85,B 0,C 180,E1 -17948.13,E2 -17948.13} C_VEL
LIN {X 0,Y 268.23,Z 369.925,A -85,B 0,C 180,E1 -17950.924,E2 -17950.924} C_VEL
LIN {X 0,Y 268.599,Z 369.199,A -85,B 0,C 180,E1 -17952.894,E2 -17952.894} C_VEL
LIN {X 0,Y 269.181,Z 367.51,A -85,B 0,C 180,E1 -17955.177,E2 -17955.177} C_VEL
LIN {X 0,Y 269.974,Z 364.918,A -85,B 0,C 180,E1 -17957.404,E2 -17957.404} C_VEL
LIN {X 0,Y 271.34,Z 360.29,A -85,B 0,C 180,E1 -17960.174,E2 -17960.174} C_VEL
LIN {X 0,Y 272.618,Z 355.613,A -85,B 0,C 180,E1 -17962.255,E2 -17962.255} C_VEL
LIN {X 0,Y 274.5,Z 348.796,A -85,B 0,C 180,E1 -17964.627,E2 -17964.627} C_VEL
LIN {X 0,Y 276.711,Z 340.266,A -85,B 0,C 180,E1 -17966.946,E2 -17966.946} C_VEL
LIN {X 0,Y 278.986,Z 331.031,A -85,B 0,C 180,E1 -17968.928,E2 -17968.928} C_VEL
LIN {X 0,Y 281.123,Z 321.174,A -85,B 0,C 180,E1 -17970.613,E2 -17970.613} C_VEL
LIN {X 0,Y 283.351,Z 309.947,A -85,B 0,C 180,E1 -17972.131,E2 -17972.131} C_VEL
LIN {X 0,Y 285.096,Z 299.066,A -85,B 0,C 180,E1 -17973.293,E2 -17973.293} C_VEL
LIN {X 0,Y 286.545,Z 286.973,A -85,B 0,C 180,E1 -17974.286,E2 -17974.286} C_VEL
LIN {X 0,Y 287.675,Z 274.27,A -85,B 0,C 180,E1 -17975.036,E2 -17975.036} C_VEL
LIN {X 0,Y 288.589,Z 260.736,A -85,B 0,C 180,E1 -17975.519,E2 -17975.519} C_VEL
LIN {X 0,Y 291.097,Z 200.362,A -85,B 0,C 180,E1 -17977.193,E2 -17977.193} C_VEL
LIN {X 0,Y 285.934,Z 188.535,A -85,B 0,C 180,E1 -17978.366,E2 -17978.366} C_VEL
LIN {X 0,Y 278.239,Z 173.975,A -85,B 0,C 180,E1 -17980.134,E2 -17980.134} C_VEL
LIN {X 0,Y 274.686,Z 168.097,A -85,B 0,C 180,E1 -17980.981,E2 -17980.981} C_VEL
LIN {X 0,Y 272.62,Z 165.288,A -85,B 0,C 180,E1 -17981.469,E2 -17981.469} C_VEL
LIN {X 0,Y 270.025,Z 163.294,A -85,B 0,C 180,E1 -17982.039,E2 -17982.039} C_VEL
LIN {X 0,Y 267.27,Z 161.985,A -85,B 0,C 180,E1 -17982.658,E2 -17982.658} C_VEL
LIN {X 0,Y 264.238,Z 161.154,A -85,B 0,C 180,E1 -17983.63,E2 -17983.63} C_VEL
LIN {X 0,Y 263.329,Z 160.689,A -85,B 0,C 180,E1 -17984.405,E2 -17984.405} C_VEL
LIN {X 0,Y 263.325,Z 160.684,A -85,B 0,C 180,E1 -17984.479,E2 -17984.479} C_VEL
LIN {X 0,Y 263.357,Z 160.68,A -85,B 0,C 180,E1 -17989.235,E2 -17989.235} C_VEL
LIN {X 0,Y 263.531,Z 160.657,A -85,B 0,C 180,E1 -17992.338,E2 -17992.338} C_VEL
LIN {X 0,Y 263.738,Z 160.626,A -85,B 0,C 180,E1 -17998.474,E2 -17998.474} C_VEL
LIN {X 0,Y 263.736,Z 160.633,A -85,B 0,C 180,E1 -18001.528,E2 -18001.528} C_VEL
LIN {X 0,Y 263.532,Z 160.647,A -85,B 0,C 180,E1 -18007.664,E2 -18007.664} C_VEL
LIN {X 0,Y 263.332,Z 160.669,A -85,B 0,C 180,E1 -18010.768,E2 -18010.768} C_VEL
LIN {X 0,Y 263.293,Z 160.675,A -85,B 0,C 180,E1 -18015.482,E2 -18015.482} C_VEL
LIN {X 0,Y 263.204,Z 160.691,A -85,B 0,C 180,E1 -18020.312,E2 -18020.312} C_VEL
LIN {X 0,Y 263.125,Z 160.708,A -85,B 0,C 180,E1 -18025.301,E2 -18025.301} C_VEL
LIN {X 0,Y 263.123,Z 160.703,A -85,B 0,C 180,E1 -18028.737,E2 -18028.737} C_VEL
LIN {X 0,Y 263.131,Z 160.701,A -85,B 0,C 180,E1 -18032.289,E2 -18032.289} C_VEL
LIN {X 0,Y 263.183,Z 160.704,A -85,B 0,C 180,E1 -18036.762,E2 -18036.762} C_VEL
LIN {X 0,Y 263.096,Z 160.714,A -85,B 0,C 180,E1 -18039.875,E2 -18039.875} C_VEL
LIN {X 0,Y 263.081,Z 160.713,A -85,B 0,C 180,E1 -18043.994,E2 -18043.994} C_VEL
LIN {X 0,Y 263.114,Z 160.75,A -85,B 0,C 180,E1 -18047.572,E2 -18047.572} C_VEL
LIN {X 0,Y 265.472,Z 168.597,A -85,B 0,C 180,E1 -18051.35,E2 -18051.35} C_VEL
LIN {X 0,Y 267.556,Z 176.318,A -85,B 0,C 180,E1 -18054.697,E2 -18054.697} C_VEL
LIN {X 0,Y 268.104,Z 178.555,A -85,B 0,C 180,E1 -18055.558,E2 -18055.558} C_VEL
LIN {X 0,Y 270.456,Z 183.078,A -85,B 0,C 180,E1 -18056.185,E2 -18056.185} C_VEL
LIN {X 0,Y 276.978,Z 196.368,A -85,B 0,C 180,E1 -18057.844,E2 -18057.844} C_VEL
LIN {X 0,Y 279.706,Z 202.985,A -85,B 0,C 180,E1 -18058.531,E2 -18058.531} C_VEL
LIN {X 0,Y 282.777,Z 222.084,A -85,B 0,C 180,E1 -18059.69,E2 -18059.69} C_VEL
LIN {X 0,Y 284.101,Z 234.362,A -85,B 0,C 180,E1 -18060.316,E2 -18060.316} C_VEL
LIN {X 0,Y 281.548,Z 289.173,A -85,B 0,C 180,E1 -18061.89,E2 -18061.89} C_VEL
LIN {X 0,Y 280.14,Z 303.088,A -85,B 0,C 180,E1 -18062.549,E2 -18062.549} C_VEL
LIN {X 0,Y 278.487,Z 315.108,A -85,B 0,C 180,E1 -18063.387,E2 -18063.387} C_VEL
LIN {X 0,Y 276.228,Z 327.633,A -85,B 0,C 180,E1 -18064.573,E2 -18064.573} C_VEL
LIN {X 0,Y 273.913,Z 338.865,A -85,B 0,C 180,E1 -18065.963,E2 -18065.963} C_VEL
LIN {X 0,Y 271.537,Z 349.076,A -85,B 0,C 180,E1 -18067.556,E2 -18067.556} C_VEL
LIN {X 0,Y 269.209,Z 358.308,A -85,B 0,C 180,E1 -18069.363,E2 -18069.363} C_VEL
LIN {X 0,Y 266.949,Z 367.338,A -85,B 0,C 180,E1 -18071.582,E2 -18071.582} C_VEL
LIN {X 0,Y 265.075,Z 374.659,A -85,B 0,C 180,E1 -18073.835,E2 -18073.835} C_VEL
LIN {X 0,Y 263.433,Z 380.566,A -85,B 0,C 180,E1 -18076.106,E2 -18076.106} C_VEL
LIN {X 0,Y 262.315,Z 385.251,A -85,B 0,C 180,E1 -18078.407,E2 -18078.407} C_VEL
LIN {X 0,Y 261.604,Z 388.849,A -85,B 0,C 180,E1 -18080.723,E2 -18080.723} C_VEL
LIN {X 0,Y 261.299,Z 390.67,A -85,B 0,C 180,E1 -18082.27,E2 -18082.27} C_VEL
LIN {X 0,Y 261.088,Z 392.802,A -85,B 0,C 180,E1 -18084.862,E2 -18084.862} C_VEL
LIN {X 0,Y 261.137,Z 393.705,A -85,B 0,C 180,E1 -18086.914,E2 -18086.914} C_VEL
LIN {X 0,Y 261.195,Z 393.874,A -85,B 0,C 180,E1 -18088.457,E2 -18088.457} C_VEL
LIN {X 0,Y 261.248,Z 393.641,A -85,B 0,C 180,E1 -18089.999,E2 -18089.999} C_VEL
LIN {X 0,Y 261.207,Z 393.002,A -85,B 0,C 180,E1 -18091.541,E2 -18091.541} C_VEL
LIN {X 0,Y 261.204,Z 391.95,A -85,B 0,C 180,E1 -18093.084,E2 -18093.084} C_VEL
LIN {X 0,Y 261.177,Z 389.581,A -85,B 0,C 180,E1 -18095.35,E2 -18095.35} C_VEL
LIN {X 0,Y 261.337,Z 386.038,A -85,B 0,C 180,E1 -18097.727,E2 -18097.727} C_VEL
LIN {X 0,Y 261.728,Z 381.424,A -85,B 0,C 180,E1 -18100.051,E2 -18100.051} C_VEL
LIN {X 0,Y 262.564,Z 374.383,A -85,B 0,C 180,E1 -18102.757,E2 -18102.757} C_VEL
LIN {X 0,Y 263.752,Z 366.745,A -85,B 0,C 180,E1 -18105.057,E2 -18105.057} C_VEL
LIN {X 0,Y 264.94,Z 358.92,A -85,B 0,C 180,E1 -18106.965,E2 -18106.965} C_VEL
LIN {X 0,Y 266.39,Z 349.346,A -85,B 0,C 180,E1 -18108.855,E2 -18108.855} C_VEL
LIN {X 0,Y 268.064,Z 338.75,A -85,B 0,C 180,E1 -18110.527,E2 -18110.527} C_VEL
LIN {X 0,Y 269.719,Z 326.965,A -85,B 0,C 180,E1 -18111.997,E2 -18111.997} C_VEL
LIN {X 0,Y 271.243,Z 314.43,A -85,B 0,C 180,E1 -18113.172,E2 -18113.172} C_VEL
LIN {X 0,Y 272.516,Z 301.365,A -85,B 0,C 180,E1 -18114.065,E2 -18114.065} C_VEL
LIN {X 0,Y 273.364,Z 288.573,A -85,B 0,C 180,E1 -18114.639,E2 -18114.639} C_VEL
LIN {X 0,Y 275.128,Z 230.161,A -85,B 0,C 180,E1 -18116.304,E2 -18116.304} C_VEL
LIN {X 0,Y 269.421,Z 187.436,A -85,B 0,C 180,E1 -18118.118,E2 -18118.118} C_VEL
LIN {X 0,Y 267.614,Z 181.587,A -85,B 0,C 180,E1 -18118.487,E2 -18118.487} C_VEL
LIN {X 0,Y 265.392,Z 170.857,A -85,B 0,C 180,E1 -18122.068,E2 -18122.068} C_VEL
LIN {X 0,Y 263.251,Z 160.693,A -85,B 0,C 180,E1 -18125.639,E2 -18125.639} C_VEL
LIN {X 0,Y 263.106,Z 160.715,A -85,B 0,C 180,E1 -18129.871,E2 -18129.871} C_VEL
LIN {X 0,Y 263.123,Z 160.712,A -85,B 0,C 180,E1 -18133.983,E2 -18133.983} C_VEL
LIN {X 0,Y 263.124,Z 160.707,A -85,B 0,C 180,E1 -18138.405,E2 -18138.405} C_VEL
LIN {X 0,Y 263.182,Z 160.703,A -85,B 0,C 180,E1 -18143.236,E2 -18143.236} C_VEL
LIN {X 0,Y 263.167,Z 160.704,A -85,B 0,C 180,E1 -18145.887,E2 -18145.887} C_VEL
LIN {X 0,Y 263.15,Z 160.705,A -85,B 0,C 180,E1 -18149.506,E2 -18149.506} C_VEL
LIN {X 0,Y 263.193,Z 160.7,A -85,B 0,C 180,E1 -18153.002,E2 -18153.002} C_VEL
LIN {X 0,Y 263.182,Z 160.696,A -85,B 0,C 180,E1 -18156.386,E2 -18156.386} C_VEL
LIN {X 0,Y 263.249,Z 160.693,A -85,B 0,C 180,E1 -18159.691,E2 -18159.691} C_VEL
LIN {X 0,Y 263.308,Z 160.681,A -85,B 0,C 180,E1 -18164.519,E2 -18164.519} C_VEL
LIN {X 0,Y 263.372,Z 160.678,A -85,B 0,C 180,E1 -18169.233,E2 -18169.233} C_VEL
LIN {X 0,Y 263.568,Z 160.646,A -85,B 0,C 180,E1 -18172.337,E2 -18172.337} C_VEL
LIN {X 0,Y 263.75,Z 160.63,A -85,B 0,C 180,E1 -18178.472,E2 -18178.472} C_VEL
LIN {X 0,Y 263.749,Z 160.623,A -85,B 0,C 180,E1 -18181.526,E2 -18181.526} C_VEL
LIN {X 0,Y 263.567,Z 160.652,A -85,B 0,C 180,E1 -18187.661,E2 -18187.661} C_VEL
LIN {X 0,Y 263.371,Z 160.676,A -85,B 0,C 180,E1 -18190.765,E2 -18190.765} C_VEL
LIN {X 0,Y 263.347,Z 160.674,A -85,B 0,C 180,E1 -18195.477,E2 -18195.477} C_VEL
LIN {X 0,Y 263.26,Z 160.693,A -85,B 0,C 180,E1 -18200.306,E2 -18200.306} C_VEL
LIN {X 0,Y 263.208,Z 160.685,A -85,B 0,C 180,E1 -18205.29,E2 -18205.29} C_VEL
LIN {X 0,Y 263.175,Z 160.699,A -85,B 0,C 180,E1 -18208.729,E2 -18208.729} C_VEL
LIN {X 0,Y 263.129,Z 160.707,A -85,B 0,C 180,E1 -18212.288,E2 -18212.288} C_VEL
LIN {X 0,Y 263.185,Z 160.694,A -85,B 0,C 180,E1 -18215.977,E2 -18215.977} C_VEL
LIN {X 0,Y 263.197,Z 160.698,A -85,B 0,C 180,E1 -18219.855,E2 -18219.855} C_VEL
LIN {X 0,Y 263.186,Z 160.699,A -85,B 0,C 180,E1 -18223.969,E2 -18223.969} C_VEL
LIN {X 0,Y 263.21,Z 160.696,A -85,B 0,C 180,E1 -18228.384,E2 -18228.384} C_VEL
LIN {X 0,Y 263.184,Z 160.7,A -85,B 0,C 180,E1 -18232.108,E2 -18232.108} C_VEL
LIN {X 0,Y 263.179,Z 160.702,A -85,B 0,C 180,E1 -18235.891,E2 -18235.891} C_VEL
LIN {X 0,Y 263.146,Z 160.708,A -85,B 0,C 180,E1 -18239.507,E2 -18239.507} C_VEL
LIN {X 0,Y 263.188,Z 160.7,A -85,B 0,C 180,E1 -18243.003,E2 -18243.003} C_VEL
LIN {X 0,Y 263.179,Z 160.7,A -85,B 0,C 180,E1 -18246.388,E2 -18246.388} C_VEL
LIN {X 0,Y 263.259,Z 160.693,A -85,B 0,C 180,E1 -18249.694,E2 -18249.694} C_VEL
LIN {X 0,Y 263.347,Z 160.681,A -85,B 0,C 180,E1 -18254.523,E2 -18254.523} C_VEL
LIN {X 0,Y 263.37,Z 160.682,A -85,B 0,C 180,E1 -18259.235,E2 -18259.235} C_VEL
LIN {X 0,Y 263.569,Z 160.653,A -85,B 0,C 180,E1 -18262.339,E2 -18262.339} C_VEL
LIN {X 0,Y 263.748,Z 160.631,A -85,B 0,C 180,E1 -18268.474,E2 -18268.474} C_VEL
LIN {X 0,Y 263.749,Z 160.631,A -85,B 0,C 180,E1 -18271.528,E2 -18271.528} C_VEL
LIN {X 0,Y 263.567,Z 160.653,A -85,B 0,C 180,E1 -18277.663,E2 -18277.663} C_VEL
LIN {X 0,Y 263.548,Z 160.657,A -85,B 0,C 180,E1 -18279.256,E2 -18279.256} C_VEL
LIN {X 0,Y 265.248,Z 165.376,A -85,B 0,C 180,E1 -18279.605,E2 -18279.605} C_VEL
LIN {X 0,Y 271.342,Z 180.391,A -85,B 0,C 180,E1 -18280.641,E2 -18280.641} C_VEL
LIN {X 0,Y 276.183,Z 194.221,A -85,B 0,C 180,E1 -18281.483,E2 -18281.483} C_VEL
LIN {X 0,Y 273.646,Z 267.131,A -85,B 0,C 180,E1 -18283.555,E2 -18283.555} C_VEL
LIN {X 0,Y 272.788,Z 280.276,A -85,B 0,C 180,E1 -18284.216,E2 -18284.216} C_VEL
LIN {X 0,Y 271.852,Z 292.908,A -85,B 0,C 180,E1 -18285.158,E2 -18285.158} C_VEL
LIN {X 0,Y 270.479,Z 305.83,A -85,B 0,C 180,E1 -18286.474,E2 -18286.474} C_VEL
LIN {X 0,Y 269.012,Z 316.607,A -85,B 0,C 180,E1 -18287.878,E2 -18287.878} C_VEL
LIN {X 0,Y 267.513,Z 326.677,A -85,B 0,C 180,E1 -18289.519,E2 -18289.519} C_VEL
LIN {X 0,Y 266.169,Z 335.456,A -85,B 0,C 180,E1 -18291.289,E2 -18291.289} C_VEL
LIN {X 0,Y 264.762,Z 344.204,A -85,B 0,C 180,E1 -18293.465,E2 -18293.465} C_VEL
LIN {X 0,Y 263.651,Z 351.337,A -85,B 0,C 180,E1 -18295.67,E2 -18295.67} C_VEL
LIN {X 0,Y 262.663,Z 357.358,A -85,B 0,C 180,E1 -18297.999,E2 -18297.999} C_VEL
LIN {X 0,Y 261.859,Z 362.858,A -85,B 0,C 180,E1 -18300.815,E2 -18300.815} C_VEL
LIN {X 0,Y 261.299,Z 366.635,A -85,B 0,C 180,E1 -18303.512,E2 -18303.512} C_VEL
LIN {X 0,Y 260.959,Z 369.145,A -85,B 0,C 180,E1 -18306.335,E2 -18306.335} C_VEL
LIN {X 0,Y 260.947,Z 370.171,A -85,B 0,C 180,E1 -18308.645,E2 -18308.645} C_VEL
LIN {X 0,Y 261.158,Z 370.266,A -85,B 0,C 180,E1 -18311.107,E2 -18311.107} C_VEL
LIN {X 0,Y 261.64,Z 369.368,A -85,B 0,C 180,E1 -18313.511,E2 -18313.511} C_VEL
LIN {X 0,Y 262.447,Z 367.061,A -85,B 0,C 180,E1 -18316.306,E2 -18316.306} C_VEL
LIN {X 0,Y 263.305,Z 364.479,A -85,B 0,C 180,E1 -18318.364,E2 -18318.364} C_VEL
LIN {X 0,Y 264.68,Z 359.971,A -85,B 0,C 180,E1 -18320.958,E2 -18320.958} C_VEL
LIN {X 0,Y 266.482,Z 353.931,A -85,B 0,C 180,E1 -18323.551,E2 -18323.551} C_VEL
LIN {X 0,Y 268.257,Z 347.795,A -85,B 0,C 180,E1 -18325.615,E2 -18325.615} C_VEL
LIN {X 0,Y 270.346,Z 340.257,A -85,B 0,C 180,E1 -18327.661,E2 -18327.661} C_VEL
LIN {X 0,Y 272.76,Z 330.827,A -85,B 0,C 180,E1 -18329.697,E2 -18329.697} C_VEL
LIN {X 0,Y 275.097,Z 320.615,A -85,B 0,C 180,E1 -18331.447,E2 -18331.447} C_VEL
LIN {X 0,Y 277.371,Z 309.382,A -85,B 0,C 180,E1 -18332.968,E2 -18332.968} C_VEL
LIN {X 0,Y 279.223,Z 297.982,A -85,B 0,C 180,E1 -18334.169,E2 -18334.169} C_VEL
LIN {X 0,Y 280.789,Z 284.986,A -85,B 0,C 180,E1 -18335.214,E2 -18335.214} C_VEL
LIN {X 0,Y 281.872,Z 272.819,A -85,B 0,C 180,E1 -18335.904,E2 -18335.904} C_VEL
LIN {X 0,Y 282.818,Z 256.596,A -85,B 0,C 180,E1 -18336.445,E2 -18336.445} C_VEL
LIN {X 0,Y 285.364,Z 202.69,A -85,B 0,C 180,E1 -18337.954,E2 -18337.954} C_VEL
LIN {X 0,Y 279.994,Z 190.549,A -85,B 0,C 180,E1 -18339.223,E2 -18339.223} C_VEL
LIN {X 0,Y 273.259,Z 177.841,A -85,B 0,C 180,E1 -18340.858,E2 -18340.858} C_VEL
LIN {X 0,Y 267.969,Z 169.092,A -85,B 0,C 180,E1 -18342.2,E2 -18342.2} C_VEL
LIN {X 0,Y 264.826,Z 164.328,A -85,B 0,C 180,E1 -18343.028,E2 -18343.028} C_VEL
LIN {X 0,Y 263.55,Z 161.962,A -85,B 0,C 180,E1 -18343.419,E2 -18343.419} C_VEL
LIN {X 0,Y 263.309,Z 160.686,A -85,B 0,C 180,E1 -18344.155,E2 -18344.155} C_VEL
LIN {X 0,Y 263.325,Z 160.684,A -85,B 0,C 180,E1 -18344.479,E2 -18344.479} C_VEL
LIN {X 0,Y 262.726,Z 160.765,A -85,B 0,C 180,E1 -18345.756,E2 -18345.756} C_VEL
LIN {X 0,Y 259.929,Z 161.112,A -85,B 0,C 180,E1 -18347.838,E2 -18347.838} C_VEL
LIN {X 0,Y 257.526,Z 161.411,A -85,B 0,C 180,E1 -18349.532,E2 -18349.532} C_VEL
LIN {X 0,Y 256.507,Z 161.54,A -85,B 0,C 180,E1 -18350.845,E2 -18350.845} C_VEL
LIN {X 0,Y 256.432,Z 161.542,A -85,B 0,C 180,E1 -18351.289,E2 -18351.289} C_VEL
LIN {X 0,Y 256.459,Z 161.543,A -85,B 0,C 180,E1 -18353.708,E2 -18353.708} C_VEL
LIN {X 0,Y 256.701,Z 161.503,A -85,B 0,C 180,E1 -18358.432,E2 -18358.432} C_VEL
LIN {X 0,Y 256.699,Z 161.508,A -85,B 0,C 180,E1 -18361.57,E2 -18361.57} C_VEL
LIN {X 0,Y 256.46,Z 161.528,A -85,B 0,C 180,E1 -18366.294,E2 -18366.294} C_VEL
LIN {X 0,Y 256.407,Z 161.543,A -85,B 0,C 180,E1 -18369.467,E2 -18369.467} C_VEL
LIN {X 0,Y 256.2,Z 161.562,A -85,B 0,C 180,E1 -18374.294,E2 -18374.294} C_VEL
LIN {X 0,Y 256.146,Z 161.578,A -85,B 0,C 180,E1 -18377.567,E2 -18377.567} C_VEL
LIN {X 0,Y 256.118,Z 161.58,A -85,B 0,C 180,E1 -18381.093,E2 -18381.093} C_VEL
LIN {X 0,Y 256.087,Z 161.583,A -85,B 0,C 180,E1 -18385.087,E2 -18385.087} C_VEL
LIN {X 0,Y 256.081,Z 161.579,A -85,B 0,C 180,E1 -18388.569,E2 -18388.569} C_VEL
LIN {X 0,Y 256.075,Z 161.577,A -85,B 0,C 180,E1 -18391.7,E2 -18391.7} C_VEL
LIN {X 0,Y 256.086,Z 161.578,A -85,B 0,C 180,E1 -18395.193,E2 -18395.193} C_VEL
LIN {X 0,Y 256.117,Z 161.581,A -85,B 0,C 180,E1 -18397.27,E2 -18397.27} C_VEL
LIN {X 0,Y 256.023,Z 161.589,A -85,B 0,C 180,E1 -18401.211,E2 -18401.211} C_VEL
LIN {X 0,Y 256.049,Z 161.593,A -85,B 0,C 180,E1 -18405.841,E2 -18405.841} C_VEL
LIN {X 0,Y 256.064,Z 161.596,A -85,B 0,C 180,E1 -18406.147,E2 -18406.147} C_VEL
LIN {X 0,Y 258.513,Z 169.677,A -85,B 0,C 180,E1 -18410.303,E2 -18410.303} C_VEL
LIN {X 0,Y 260.847,Z 177.961,A -85,B 0,C 180,E1 -18414.07,E2 -18414.07} C_VEL
LIN {X 0,Y 263.117,Z 182.387,A -85,B 0,C 180,E1 -18414.732,E2 -18414.732} C_VEL
LIN {X 0,Y 268.767,Z 193.268,A -85,B 0,C 180,E1 -18416.278,E2 -18416.278} C_VEL
LIN {X 0,Y 273.827,Z 204.367,A -85,B 0,C 180,E1 -18417.612,E2 -18417.612} C_VEL
LIN {X 0,Y 274.78,Z 208.147,A -85,B 0,C 180,E1 -18417.919,E2 -18417.919} C_VEL
LIN {X 0,Y 277.612,Z 227.447,A -85,B 0,C 180,E1 -18419.089,E2 -18419.089} C_VEL
LIN {X 0,Y 278.362,Z 234.874,A -85,B 0,C 180,E1 -18419.473,E2 -18419.473} C_VEL
LIN {X 0,Y 275.674,Z 289.429,A -85,B 0,C 180,E1 -18421.079,E2 -18421.079} C_VEL
LIN {X 0,Y 274.216,Z 303.09,A -85,B 0,C 180,E1 -18421.747,E2 -18421.747} C_VEL
LIN {X 0,Y 272.569,Z 314.438,A -85,B 0,C 180,E1 -18422.554,E2 -18422.554} C_VEL
LIN {X 0,Y 270.216,Z 327.004,A -85,B 0,C 180,E1 -18423.758,E2 -18423.758} C_VEL
LIN {X 0,Y 268.12,Z 336.963,A -85,B 0,C 180,E1 -18424.996,E2 -18424.996} C_VEL
LIN {X 0,Y 265.575,Z 347.454,A -85,B 0,C 180,E1 -18426.611,E2 -18426.611} C_VEL
LIN {X 0,Y 263.051,Z 356.97,A -85,B 0,C 180,E1 -18428.446,E2 -18428.446} C_VEL
LIN {X 0,Y 260.928,Z 364.807,A -85,B 0,C 180,E1 -18430.325,E2 -18430.325} C_VEL
LIN {X 0,Y 258.778,Z 372.504,A -85,B 0,C 180,E1 -18432.617,E2 -18432.617} C_VEL
LIN {X 0,Y 257.071,Z 378.741,A -85,B 0,C 180,E1 -18434.946,E2 -18434.946} C_VEL
LIN {X 0,Y 255.625,Z 383.726,A -85,B 0,C 180,E1 -18437.293,E2 -18437.293} C_VEL
LIN {X 0,Y 254.761,Z 387.6,A -85,B 0,C 180,E1 -18439.669,E2 -18439.669} C_VEL
LIN {X 0,Y 254.24,Z 390.47,A -85,B 0,C 180,E1 -18442.054,E2 -18442.054} C_VEL
LIN {X 0,Y 253.977,Z 392.835,A -85,B 0,C 180,E1 -18445.237,E2 -18445.237} C_VEL
LIN {X 0,Y 254.047,Z 393.395,A -85,B 0,C 180,E1 -18446.827,E2 -18446.827} C_VEL
LIN {X 0,Y 254.119,Z 393.531,A -85,B 0,C 180,E1 -18448.414,E2 -18448.414} C_VEL
LIN {X 0,Y 254.17,Z 393.268,A -85,B 0,C 180,E1 -18449.999,E2 -18449.999} C_VEL
LIN {X 0,Y 254.133,Z 392.601,A -85,B 0,C 180,E1 -18451.584,E2 -18451.584} C_VEL
LIN {X 0,Y 254.113,Z 391.49,A -85,B 0,C 180,E1 -18453.17,E2 -18453.17} C_VEL
LIN {X 0,Y 254.088,Z 389.337,A -85,B 0,C 180,E1 -18455.276,E2 -18455.276} C_VEL
LIN {X 0,Y 254.289,Z 385.456,A -85,B 0,C 180,E1 -18457.942,E2 -18457.942} C_VEL
LIN {X 0,Y 254.701,Z 380.755,A -85,B 0,C 180,E1 -18460.331,E2 -18460.331} C_VEL
LIN {X 0,Y 255.415,Z 374.758,A -85,B 0,C 180,E1 -18462.716,E2 -18462.716} C_VEL
LIN {X 0,Y 256.647,Z 367.272,A -85,B 0,C 180,E1 -18465.078,E2 -18465.078} C_VEL
LIN {X 0,Y 257.858,Z 359.616,A -85,B 0,C 180,E1 -18467.036,E2 -18467.036} C_VEL
LIN {X 0,Y 259.321,Z 350.33,A -85,B 0,C 180,E1 -18468.978,E2 -18468.978} C_VEL
LIN {X 0,Y 261.016,Z 340.022,A -85,B 0,C 180,E1 -18470.694,E2 -18470.694} C_VEL
LIN {X 0,Y 262.682,Z 328.603,A -85,B 0,C 180,E1 -18472.203,E2 -18472.203} C_VEL
LIN {X 0,Y 264.206,Z 316.802,A -85,B 0,C 180,E1 -18473.411,E2 -18473.411} C_VEL
LIN {X 0,Y 265.562,Z 303.931,A -85,B 0,C 180,E1 -18474.373,E2 -18474.373} C_VEL
LIN {X 0,Y 266.521,Z 290.732,A -85,B 0,C 180,E1 -18475.047,E2 -18475.047} C_VEL
LIN {X 0,Y 268.582,Z 232.215,A -85,B 0,C 180,E1 -18476.765,E2 -18476.765} C_VEL
LIN {X 0,Y 263.09,Z 189.697,A -85,B 0,C 180,E1 -18478.614,E2 -18478.614} C_VEL
LIN {X 0,Y 260.326,Z 181.212,A -85,B 0,C 180,E1 -18479.184,E2 -18479.184} C_VEL
LIN {X 0,Y 258.311,Z 171.623,A -85,B 0,C 180,E1 -18482.494,E2 -18482.494} C_VEL
LIN {X 0,Y 256.182,Z 161.573,A -85,B 0,C 180,E1 -18486.143,E2 -18486.143} C_VEL
LIN {X 0,Y 256.061,Z 161.593,A -85,B 0,C 180,E1 -18489.779,E2 -18489.779} C_VEL
LIN {X 0,Y 256.062,Z 161.591,A -85,B 0,C 180,E1 -18493.326,E2 -18493.326} C_VEL
LIN {X 0,Y 256.072,Z 161.588,A -85,B 0,C 180,E1 -18497.818,E2 -18497.818} C_VEL
LIN {X 0,Y 256.071,Z 161.586,A -85,B 0,C 180,E1 -18500.857,E2 -18500.857} C_VEL
LIN {X 0,Y 256.108,Z 161.582,A -85,B 0,C 180,E1 -18504.81,E2 -18504.81} C_VEL
LIN {X 0,Y 256.092,Z 161.584,A -85,B 0,C 180,E1 -18508.571,E2 -18508.571} C_VEL
LIN {X 0,Y 256.142,Z 161.577,A -85,B 0,C 180,E1 -18512.195,E2 -18512.195} C_VEL
LIN {X 0,Y 256.166,Z 161.571,A -85,B 0,C 180,E1 -18515.698,E2 -18515.698} C_VEL
LIN {X 0,Y 256.16,Z 161.577,A -85,B 0,C 180,E1 -18519.103,E2 -18519.103} C_VEL
LIN {X 0,Y 256.243,Z 161.56,A -85,B 0,C 180,E1 -18524.081,E2 -18524.081} C_VEL
LIN {X 0,Y 256.287,Z 161.562,A -85,B 0,C 180,E1 -18527.327,E2 -18527.327} C_VEL
LIN {X 0,Y 256.478,Z 161.534,A -85,B 0,C 180,E1 -18530.559,E2 -18530.559} C_VEL
LIN {X 0,Y 256.483,Z 161.531,A -85,B 0,C 180,E1 -18533.707,E2 -18533.707} C_VEL
LIN {X 0,Y 256.712,Z 161.507,A -85,B 0,C 180,E1 -18538.43,E2 -18538.43} C_VEL
LIN {X 0,Y 256.712,Z 161.498,A -85,B 0,C 180,E1 -18541.568,E2 -18541.568} C_VEL
LIN {X 0,Y 256.535,Z 161.528,A -85,B 0,C 180,E1 -18547.872,E2 -18547.872} C_VEL
LIN {X 0,Y 256.306,Z 161.553,A -85,B 0,C 180,E1 -18551.065,E2 -18551.065} C_VEL
LIN {X 0,Y 256.296,Z 161.553,A -85,B 0,C 180,E1 -18555.914,E2 -18555.914} C_VEL
LIN {X 0,Y 256.163,Z 161.574,A -85,B 0,C 180,E1 -18560.894,E2 -18560.894} C_VEL
LIN {X 0,Y 256.188,Z 161.559,A -85,B 0,C 180,E1 -18565.14,E2 -18565.14} C_VEL
LIN {X 0,Y 256.109,Z 161.578,A -85,B 0,C 180,E1 -18569.599,E2 -18569.599} C_VEL
LIN {X 0,Y 256.08,Z 161.581,A -85,B 0,C 180,E1 -18573.29,E2 -18573.29} C_VEL
LIN {X 0,Y 256.136,Z 161.569,A -85,B 0,C 180,E1 -18577.278,E2 -18577.278} C_VEL
LIN {X 0,Y 256.159,Z 161.573,A -85,B 0,C 180,E1 -18581.182,E2 -18581.182} C_VEL
LIN {X 0,Y 256.112,Z 161.577,A -85,B 0,C 180,E1 -18585.516,E2 -18585.516} C_VEL
LIN {X 0,Y 256.159,Z 161.573,A -85,B 0,C 180,E1 -18588.818,E2 -18588.818} C_VEL
LIN {X 0,Y 256.151,Z 161.574,A -85,B 0,C 180,E1 -18592.872,E2 -18592.872} C_VEL
LIN {X 0,Y 256.08,Z 161.583,A -85,B 0,C 180,E1 -18596.71,E2 -18596.71} C_VEL
LIN {X 0,Y 256.134,Z 161.58,A -85,B 0,C 180,E1 -18601.405,E2 -18601.405} C_VEL
LIN {X 0,Y 256.162,Z 161.577,A -85,B 0,C 180,E1 -18605.7,E2 -18605.7} C_VEL
LIN {X 0,Y 256.162,Z 161.577,A -85,B 0,C 180,E1 -18609.105,E2 -18609.105} C_VEL
LIN {X 0,Y 256.296,Z 161.559,A -85,B 0,C 180,E1 -18614.086,E2 -18614.086} C_VEL
LIN {X 0,Y 256.306,Z 161.561,A -85,B 0,C 180,E1 -18618.935,E2 -18618.935} C_VEL
LIN {X 0,Y 256.536,Z 161.529,A -85,B 0,C 180,E1 -18622.128,E2 -18622.128} C_VEL
LIN {X 0,Y 256.711,Z 161.508,A -85,B 0,C 180,E1 -18628.432,E2 -18628.432} C_VEL
LIN {X 0,Y 256.712,Z 161.507,A -85,B 0,C 180,E1 -18631.57,E2 -18631.57} C_VEL
LIN {X 0,Y 256.535,Z 161.529,A -85,B 0,C 180,E1 -18637.874,E2 -18637.874} C_VEL
LIN {X 0,Y 256.518,Z 161.535,A -85,B 0,C 180,E1 -18638.618,E2 -18638.618} C_VEL
LIN {X 0,Y 257.525,Z 164.427,A -85,B 0,C 180,E1 -18638.825,E2 -18638.825} C_VEL
LIN {X 0,Y 263.672,Z 179.237,A -85,B 0,C 180,E1 -18639.909,E2 -18639.909} C_VEL
LIN {X 0,Y 269.519,Z 195.626,A -85,B 0,C 180,E1 -18640.962,E2 -18640.962} C_VEL
LIN {X 0,Y 266.94,Z 267.608,A -85,B 0,C 180,E1 -18643.064,E2 -18643.064} C_VEL
LIN {X 0,Y 266.073,Z 280.465,A -85,B 0,C 180,E1 -18643.726,E2 -18643.726} C_VEL
LIN {X 0,Y 265.115,Z 293.063,A -85,B 0,C 180,E1 -18644.685,E2 -18644.685} C_VEL
LIN {X 0,Y 263.751,Z 305.522,A -85,B 0,C 180,E1 -18645.972,E2 -18645.972} C_VEL
LIN {X 0,Y 262.114,Z 317.417,A -85,B 0,C 180,E1 -18647.557,E2 -18647.557} C_VEL
LIN {X 0,Y 260.552,Z 327.456,A -85,B 0,C 180,E1 -18649.256,E2 -18649.256} C_VEL
LIN {X 0,Y 259.187,Z 336.095,A -85,B 0,C 180,E1 -18651.057,E2 -18651.057} C_VEL
LIN {X 0,Y 257.721,Z 344.806,A -85,B 0,C 180,E1 -18653.293,E2 -18653.293} C_VEL
LIN {X 0,Y 256.665,Z 351.339,A -85,B 0,C 180,E1 -18655.366,E2 -18655.366} C_VEL
LIN {X 0,Y 255.607,Z 357.68,A -85,B 0,C 180,E1 -18657.868,E2 -18657.868} C_VEL
LIN {X 0,Y 254.863,Z 362.702,A -85,B 0,C 180,E1 -18660.464,E2 -18660.464} C_VEL
LIN {X 0,Y 254.379,Z 365.868,A -85,B 0,C 180,E1 -18662.6,E2 -18662.6} C_VEL
LIN {X 0,Y 253.912,Z 368.838,A -85,B 0,C 180,E1 -18665.54,E2 -18665.54} C_VEL
LIN {X 0,Y 253.837,Z 370.066,A -85,B 0,C 180,E1 -18667.527,E2 -18667.527} C_VEL
LIN {X 0,Y 253.909,Z 370.612,A -85,B 0,C 180,E1 -18669.542,E2 -18669.542} C_VEL
LIN {X 0,Y 254.172,Z 370.508,A -85,B 0,C 180,E1 -18671.708,E2 -18671.708} C_VEL
LIN {X 0,Y 254.708,Z 369.482,A -85,B 0,C 180,E1 -18674.161,E2 -18674.161} C_VEL
LIN {X 0,Y 255.44,Z 367.555,A -85,B 0,C 180,E1 -18676.543,E2 -18676.543} C_VEL
LIN {X 0,Y 256.462,Z 364.709,A -85,B 0,C 180,E1 -18678.878,E2 -18678.878} C_VEL
LIN {X 0,Y 257.694,Z 360.939,A -85,B 0,C 180,E1 -18681.152,E2 -18681.152} C_VEL
LIN {X 0,Y 259.514,Z 355.254,A -85,B 0,C 180,E1 -18683.74,E2 -18683.74} C_VEL
LIN {X 0,Y 261.813,Z 347.844,A -85,B 0,C 180,E1 -18686.322,E2 -18686.322} C_VEL
LIN {X 0,Y 264.022,Z 340.244,A -85,B 0,C 180,E1 -18688.41,E2 -18688.41} C_VEL
LIN {X 0,Y 266.534,Z 330.763,A -85,B 0,C 180,E1 -18690.478,E2 -18690.478} C_VEL
LIN {X 0,Y 269.101,Z 320.165,A -85,B 0,C 180,E1 -18692.31,E2 -18692.31} C_VEL
LIN {X 0,Y 271.372,Z 309.392,A -85,B 0,C 180,E1 -18693.777,E2 -18693.777} C_VEL
LIN {X 0,Y 273.212,Z 298.683,A -85,B 0,C 180,E1 -18694.929,E2 -18694.929} C_VEL
LIN {X 0,Y 274.798,Z 286.38,A -85,B 0,C 180,E1 -18695.952,E2 -18695.952} C_VEL
LIN {X 0,Y 276.012,Z 273.64,A -85,B 0,C 180,E1 -18696.708,E2 -18696.708} C_VEL
LIN {X 0,Y 276.959,Z 258.382,A -85,B 0,C 180,E1 -18697.24,E2 -18697.24} C_VEL
LIN {X 0,Y 279.6,Z 204.783,A -85,B 0,C 180,E1 -18698.768,E2 -18698.768} C_VEL
LIN {X 0,Y 274.609,Z 193.515,A -85,B 0,C 180,E1 -18700.015,E2 -18700.015} C_VEL
LIN {X 0,Y 268.463,Z 181.874,A -85,B 0,C 180,E1 -18701.581,E2 -18701.581} C_VEL
LIN {X 0,Y 262.371,Z 171.618,A -85,B 0,C 180,E1 -18703.228,E2 -18703.228} C_VEL
LIN {X 0,Y 258.329,Z 165.735,A -85,B 0,C 180,E1 -18704.366,E2 -18704.366} C_VEL
LIN {X 0,Y 256.631,Z 163.11,A -85,B 0,C 180,E1 -18704.87,E2 -18704.87} C_VEL
LIN {X 0,Y 256.426,Z 162.396,A -85,B 0,C 180,E1 -18705.01,E2 -18705.01} C_VEL
LIN {X 0,Y 256.241,Z 161.571,A -85,B 0,C 180,E1 -18705.507,E2 -18705.507} C_VEL
LIN {X 0,Y 256.299,Z 161.561,A -85,B 0,C 180,E1 -18708.934,E2 -18708.934} C_VEL
LIN {X 0,Y 256.432,Z 161.542,A -85,B 0,C 180,E1 -18711.289,E2 -18711.289} C_VEL
LIN {X 0,Y 255.762,Z 161.625,A -85,B 0,C 180,E1 -18712.599,E2 -18712.599} C_VEL
LIN {X 0,Y 252.862,Z 161.987,A -85,B 0,C 180,E1 -18714.732,E2 -18714.732} C_VEL
LIN {X 0,Y 250.497,Z 162.278,A -85,B 0,C 180,E1 -18716.47,E2 -18716.47} C_VEL
LIN {X 0,Y 249.628,Z 162.391,A -85,B 0,C 180,E1 -18717.817,E2 -18717.817} C_VEL
LIN {X 0,Y 249.636,Z 162.383,A -85,B 0,C 180,E1 -18718.272,E2 -18718.272} C_VEL
LIN {X 0,Y 249.66,Z 162.384,A -85,B 0,C 180,E1 -18721.614,E2 -18721.614} C_VEL
LIN {X 0,Y 249.431,Z 162.402,A -85,B 0,C 180,E1 -18726.472,E2 -18726.472} C_VEL
LIN {X 0,Y 249.337,Z 162.42,A -85,B 0,C 180,E1 -18729.738,E2 -18729.738} C_VEL
LIN {X 0,Y 249.147,Z 162.437,A -85,B 0,C 180,E1 -18734.708,E2 -18734.708} C_VEL
LIN {X 0,Y 249.078,Z 162.455,A -85,B 0,C 180,E1 -18738.083,E2 -18738.083} C_VEL
LIN {X 0,Y 249.045,Z 162.464,A -85,B 0,C 180,E1 -18741.523,E2 -18741.523} C_VEL
LIN {X 0,Y 249.048,Z 162.462,A -85,B 0,C 180,E1 -18745.439,E2 -18745.439} C_VEL
LIN {X 0,Y 249.029,Z 162.461,A -85,B 0,C 180,E1 -18748.968,E2 -18748.968} C_VEL
LIN {X 0,Y 249.031,Z 162.458,A -85,B 0,C 180,E1 -18752.427,E2 -18752.427} C_VEL
LIN {X 0,Y 249.051,Z 162.461,A -85,B 0,C 180,E1 -18756.343,E2 -18756.343} C_VEL
LIN {X 0,Y 248.984,Z 162.469,A -85,B 0,C 180,E1 -18760.483,E2 -18760.483} C_VEL
LIN {X 0,Y 249.009,Z 162.532,A -85,B 0,C 180,E1 -18764.595,E2 -18764.595} C_VEL
LIN {X 0,Y 251.444,Z 170.474,A -85,B 0,C 180,E1 -18768.997,E2 -18768.997} C_VEL
LIN {X 0,Y 253.555,Z 177.588,A -85,B 0,C 180,E1 -18772.424,E2 -18772.424} C_VEL
LIN {X 0,Y 256.185,Z 182.238,A -85,B 0,C 180,E1 -18773.239,E2 -18773.239} C_VEL
LIN {X 0,Y 262.558,Z 194.311,A -85,B 0,C 180,E1 -18775.122,E2 -18775.122} C_VEL
LIN {X 0,Y 267.549,Z 205.025,A -85,B 0,C 180,E1 -18776.52,E2 -18776.52} C_VEL
LIN {X 0,Y 269.276,Z 209.576,A -85,B 0,C 180,E1 -18777.013,E2 -18777.013} C_VEL
LIN {X 0,Y 272.121,Z 229.86,A -85,B 0,C 180,E1 -18778.293,E2 -18778.293} C_VEL
LIN {X 0,Y 272.666,Z 235.758,A -85,B 0,C 180,E1 -18778.606,E2 -18778.606} C_VEL
LIN {X 0,Y 269.983,Z 288.468,A -85,B 0,C 180,E1 -18780.182,E2 -18780.182} C_VEL
LIN {X 0,Y 268.581,Z 301.736,A -85,B 0,C 180,E1 -18780.832,E2 -18780.832} C_VEL
LIN {X 0,Y 266.524,Z 314.934,A -85,B 0,C 180,E1 -18781.77,E2 -18781.77} C_VEL
LIN {X 0,Y 264.282,Z 326.513,A -85,B 0,C 180,E1 -18782.908,E2 -18782.908} C_VEL
LIN {X 0,Y 262.081,Z 336.499,A -85,B 0,C 180,E1 -18784.165,E2 -18784.165} C_VEL
LIN {X 0,Y 259.667,Z 345.91,A -85,B 0,C 180,E1 -18785.621,E2 -18785.621} C_VEL
LIN {X 0,Y 256.932,Z 355.601,A -85,B 0,C 180,E1 -18787.482,E2 -18787.482} C_VEL
LIN {X 0,Y 254.672,Z 363.586,A -85,B 0,C 180,E1 -18789.399,E2 -18789.399} C_VEL
LIN {X 0,Y 252.34,Z 371.6,A -85,B 0,C 180,E1 -18791.782,E2 -18791.782} C_VEL
LIN {X 0,Y 250.203,Z 378.776,A -85,B 0,C 180,E1 -18794.522,E2 -18794.522} C_VEL
LIN {X 0,Y 248.669,Z 383.685,A -85,B 0,C 180,E1 -18796.931,E2 -18796.931} C_VEL
LIN {X 0,Y 247.755,Z 387.486,A -85,B 0,C 180,E1 -18799.374,E2 -18799.374} C_VEL
LIN {X 0,Y 247.181,Z 390.281,A -85,B 0,C 180,E1 -18801.826,E2 -18801.826} C_VEL
LIN {X 0,Y 246.976,Z 391.627,A -85,B 0,C 180,E1 -18803.463,E2 -18803.463} C_VEL
LIN {X 0,Y 246.885,Z 392.572,A -85,B 0,C 180,E1 -18805.1,E2 -18805.1} C_VEL
LIN {X 0,Y 246.96,Z 393.08,A -85,B 0,C 180,E1 -18806.736,E2 -18806.736} C_VEL
LIN {X 0,Y 247.044,Z 393.189,A -85,B 0,C 180,E1 -18808.369,E2 -18808.369} C_VEL
LIN {X 0,Y 247.094,Z 392.897,A -85,B 0,C 180,E1 -18809.999,E2 -18809.999} C_VEL
LIN {X 0,Y 247.06,Z 392.194,A -85,B 0,C 180,E1 -18811.629,E2 -18811.629} C_VEL
LIN {X 0,Y 247.025,Z 391.025,A -85,B 0,C 180,E1 -18813.261,E2 -18813.261} C_VEL
LIN {X 0,Y 246.99,Z 389.117,A -85,B 0,C 180,E1 -18815.176,E2 -18815.176} C_VEL
LIN {X 0,Y 247.133,Z 386.171,A -85,B 0,C 180,E1 -18817.351,E2 -18817.351} C_VEL
LIN {X 0,Y 247.507,Z 381.799,A -85,B 0,C 180,E1 -18819.808,E2 -18819.808} C_VEL
LIN {X 0,Y 248.131,Z 376.182,A -85,B 0,C 180,E1 -18822.264,E2 -18822.264} C_VEL
LIN {X 0,Y 249.345,Z 369.165,A -85,B 0,C 180,E1 -18824.694,E2 -18824.694} C_VEL
LIN {X 0,Y 250.757,Z 360.417,A -85,B 0,C 180,E1 -18827.087,E2 -18827.087} C_VEL
LIN {X 0,Y 252.238,Z 351.224,A -85,B 0,C 180,E1 -18829.109,E2 -18829.109} C_VEL
LIN {X 0,Y 253.905,Z 341.248,A -85,B 0,C 180,E1 -18830.877,E2 -18830.877} C_VEL
LIN {X 0,Y 255.657,Z 330.222,A -85,B 0,C 180,E1 -18832.421,E2 -18832.421} C_VEL
LIN {X 0,Y 257.275,Z 317.901,A -85,B 0,C 180,E1 -18833.76,E2 -18833.76} C_VEL
LIN {X 0,Y 258.75,Z 305.008,A -85,B 0,C 180,E1 -18834.79,E2 -18834.79} C_VEL
LIN {X 0,Y 259.736,Z 292.196,A -85,B 0,C 180,E1 -18835.492,E2 -18835.492} C_VEL
LIN {X 0,Y 260.609,Z 270.714,A -85,B 0,C 180,E1 -18836.188,E2 -18836.188} C_VEL
LIN {X 0,Y 261.858,Z 231.581,A -85,B 0,C 180,E1 -18837.351,E2 -18837.351} C_VEL
LIN {X 0,Y 256.478,Z 190.831,A -85,B 0,C 180,E1 -18839.2,E2 -18839.2} C_VEL
LIN {X 0,Y 253.053,Z 180.917,A -85,B 0,C 180,E1 -18839.897,E2 -18839.897} C_VEL
LIN {X 0,Y 250.581,Z 169.124,A -85,B 0,C 180,E1 -18844.12,E2 -18844.12} C_VEL
LIN {X 0,Y 249.12,Z 162.454,A -85,B 0,C 180,E1 -18846.706,E2 -18846.706} C_VEL
LIN {X 0,Y 249.006,Z 162.47,A -85,B 0,C 180,E1 -18850.477,E2 -18850.477} C_VEL
LIN {X 0,Y 249.003,Z 162.469,A -85,B 0,C 180,E1 -18854.878,E2 -18854.878} C_VEL
LIN {X 0,Y 249.016,Z 162.467,A -85,B 0,C 180,E1 -18857.362,E2 -18857.362} C_VEL
LIN {X 0,Y 249.043,Z 162.463,A -85,B 0,C 180,E1 -18862.199,E2 -18862.199} C_VEL
LIN {X 0,Y 249.056,Z 162.462,A -85,B 0,C 180,E1 -18865.64,E2 -18865.64} C_VEL
LIN {X 0,Y 249.051,Z 162.461,A -85,B 0,C 180,E1 -18869.472,E2 -18869.472} C_VEL
LIN {X 0,Y 249.074,Z 162.46,A -85,B 0,C 180,E1 -18873.161,E2 -18873.161} C_VEL
LIN {X 0,Y 249.077,Z 162.453,A -85,B 0,C 180,E1 -18876.731,E2 -18876.731} C_VEL
LIN {X 0,Y 249.091,Z 162.455,A -85,B 0,C 180,E1 -18880.209,E2 -18880.209} C_VEL
LIN {X 0,Y 249.194,Z 162.439,A -85,B 0,C 180,E1 -18883.618,E2 -18883.618} C_VEL
LIN {X 0,Y 249.249,Z 162.437,A -85,B 0,C 180,E1 -18888.616,E2 -18888.616} C_VEL
LIN {X 0,Y 249.478,Z 162.4,A -85,B 0,C 180,E1 -18891.902,E2 -18891.902} C_VEL
LIN {X 0,Y 249.434,Z 162.415,A -85,B 0,C 180,E1 -18896.769,E2 -18896.769} C_VEL
LIN {X 0,Y 249.733,Z 162.372,A -85,B 0,C 180,E1 -18899.999,E2 -18899.999} C_VEL
LIN {X 0,Y 249.433,Z 162.408,A -85,B 0,C 180,E1 -18903.23,E2 -18903.23} C_VEL
LIN {X 0,Y 249.477,Z 162.408,A -85,B 0,C 180,E1 -18908.096,E2 -18908.096} C_VEL
LIN {X 0,Y 249.25,Z 162.431,A -85,B 0,C 180,E1 -18911.383,E2 -18911.383} C_VEL
LIN {X 0,Y 249.238,Z 162.434,A -85,B 0,C 180,E1 -18916.377,E2 -18916.377} C_VEL
LIN {X 0,Y 249.084,Z 162.454,A -85,B 0,C 180,E1 -18921.517,E2 -18921.517} C_VEL
LIN {X 0,Y 249.13,Z 162.437,A -85,B 0,C 180,E1 -18925.483,E2 -18925.483} C_VEL
LIN {X 0,Y 249.079,Z 162.453,A -85,B 0,C 180,E1 -18928.993,E2 -18928.993} C_VEL
LIN {X 0,Y 249.031,Z 162.461,A -85,B 0,C 180,E1 -18932.425,E2 -18932.425} C_VEL
LIN {X 0,Y 249.071,Z 162.45,A -85,B 0,C 180,E1 -18936.337,E2 -18936.337} C_VEL
LIN {X 0,Y 249.1,Z 162.454,A -85,B 0,C 180,E1 -18940.458,E2 -18940.458} C_VEL
LIN {X 0,Y 249.058,Z 162.453,A -85,B 0,C 180,E1 -18944.865,E2 -18944.865} C_VEL
LIN {X 0,Y 249.094,Z 162.45,A -85,B 0,C 180,E1 -18947.381,E2 -18947.381} C_VEL
LIN {X 0,Y 249.068,Z 162.461,A -85,B 0,C 180,E1 -18951.628,E2 -18951.628} C_VEL
LIN {X 0,Y 249.057,Z 162.457,A -85,B 0,C 180,E1 -18955.643,E2 -18955.643} C_VEL
LIN {X 0,Y 249.047,Z 162.464,A -85,B 0,C 180,E1 -18959.474,E2 -18959.474} C_VEL
LIN {X 0,Y 249.069,Z 162.46,A -85,B 0,C 180,E1 -18963.163,E2 -18963.163} C_VEL
LIN {X 0,Y 249.075,Z 162.457,A -85,B 0,C 180,E1 -18966.733,E2 -18966.733} C_VEL
LIN {X 0,Y 249.106,Z 162.454,A -85,B 0,C 180,E1 -18970.212,E2 -18970.212} C_VEL
LIN {X 0,Y 249.238,Z 162.441,A -85,B 0,C 180,E1 -18973.623,E2 -18973.623} C_VEL
LIN {X 0,Y 249.249,Z 162.438,A -85,B 0,C 180,E1 -18978.617,E2 -18978.617} C_VEL
LIN {X 0,Y 249.481,Z 162.409,A -85,B 0,C 180,E1 -18981.904,E2 -18981.904} C_VEL
LIN {X 0,Y 249.434,Z 162.416,A -85,B 0,C 180,E1 -18986.771,E2 -18986.771} C_VEL
LIN {X 0,Y 249.725,Z 162.377,A -85,B 0,C 180,E1 -18990.001,E2 -18990.001} C_VEL
LIN {X 0,Y 249.434,Z 162.414,A -85,B 0,C 180,E1 -18993.231,E2 -18993.231} C_VEL
LIN {X 0,Y 249.505,Z 162.481,A -85,B 0,C 180,E1 -18997.945,E2 -18997.945} C_VEL
LIN {X 0,Y 251.187,Z 166.918,A -85,B 0,C 180,E1 -18998.274,E2 -18998.274} C_VEL
LIN {X 0,Y 257.419,Z 181.658,A -85,B 0,C 180,E1 -18999.394,E2 -18999.394} C_VEL
LIN {X 0,Y 262.916,Z 196.987,A -85,B 0,C 180,E1 -19000.418,E2 -19000.418} C_VEL
LIN {X 0,Y 260.286,Z 267.549,A -85,B 0,C 180,E1 -19002.525,E2 -19002.525} C_VEL
LIN {X 0,Y 259.367,Z 281.166,A -85,B 0,C 180,E1 -19003.246,E2 -19003.246} C_VEL
LIN {X 0,Y 258.324,Z 294.129,A -85,B 0,C 180,E1 -19004.275,E2 -19004.275} C_VEL
LIN {X 0,Y 257.047,Z 305.345,A -85,B 0,C 180,E1 -19005.462,E2 -19005.462} C_VEL
LIN {X 0,Y 255.345,Z 317.326,A -85,B 0,C 180,E1 -19007.084,E2 -19007.084} C_VEL
LIN {X 0,Y 253.62,Z 328.153,A -85,B 0,C 180,E1 -19008.963,E2 -19008.963} C_VEL
LIN {X 0,Y 252.196,Z 336.742,A -85,B 0,C 180,E1 -19010.813,E2 -19010.813} C_VEL
LIN {X 0,Y 250.699,Z 345.401,A -85,B 0,C 180,E1 -19013.109,E2 -19013.109} C_VEL
LIN {X 0,Y 249.419,Z 352.932,A -85,B 0,C 180,E1 -19015.623,E2 -19015.623} C_VEL
LIN {X 0,Y 248.541,Z 358.054,A -85,B 0,C 180,E1 -19017.753,E2 -19017.753} C_VEL
LIN {X 0,Y 247.706,Z 363.522,A -85,B 0,C 180,E1 -19020.712,E2 -19020.712} C_VEL
LIN {X 0,Y 247.266,Z 366.305,A -85,B 0,C 180,E1 -19022.687,E2 -19022.687} C_VEL
LIN {X 0,Y 246.915,Z 368.417,A -85,B 0,C 180,E1 -19024.7,E2 -19024.7} C_VEL
LIN {X 0,Y 246.747,Z 370.106,A -85,B 0,C 180,E1 -19027.108,E2 -19027.108} C_VEL
